  Set speed (120.0 mm/s)
  MoveL 7621 to (504.18, 492.37, 15.4) mm, rotated rx 0 ry 90 rz 0 deg; joints [-11.231, -27.866, 111.232, -15.254, -82.736, 50.97]
  Set speed (1000.0 mm/s)
  MoveL 7622 to (504.11, 492.3, 15.4) mm, rotated rx 0 ry 90 rz 0 deg; joints [-11.226, -27.867, 111.243, -15.248, -82.744, 50.967]
  Set speed (15.0 mm/s)
  Call Extruder(0.010)
  MoveL 7623 to (504.11, 491.95, 15.4) mm, rotated rx 0 ry 90 rz 0 deg; joints [-11.194, -27.869, 111.251, -15.216, -82.75, 50.961]
  Call Extruder(0.035)
  MoveL 7624 to (504.11, 490.75, 15.4) mm, rotated rx 0 ry 90 rz 0 deg; joints [-11.084, -27.873, 111.279, -15.104, -82.77, 50.943]
  Call Extruder(0.010)
  MoveL 7625 to (504.11, 490.4, 15.4) mm, rotated rx 0 ry 90 rz 0 deg; joints [-11.052, -27.874, 111.288, -15.072, -82.776, 50.937]
  Call Extruder(0.007)
  MoveL 7626 to (504.46, 490.4, 15.4) mm, rotated rx 0 ry 90 rz 0 deg; joints [-11.046, -27.868, 111.246, -15.067, -82.741, 50.946]
  Call Extruder(0.149)
  MoveL 7627 to (509.6, 490.4, 15.4) mm, rotated rx 0 ry 90 rz 0 deg; joints [-10.955, -27.767, 110.627, -14.993, -82.238, 51.071]
  Call Extruder(0.125)
  MoveL 7628 to (509.6, 494.7, 15.4) mm, rotated rx 0 ry 90 rz 0 deg; joints [-11.345, -27.75, 110.525, -15.389, -82.169, 51.141]
  Call Extruder(0.046)
  MoveL 7629 to (508.02, 494.7, 15.4) mm, rotated rx 0 ry 90 rz 0 deg; joints [-11.374, -27.781, 110.715, -15.413, -82.323, 51.102]
  Call Extruder(0.010)
  MoveL 7630 to (507.67, 494.7, 15.4) mm, rotated rx 0 ry 90 rz 0 deg; joints [-11.38, -27.788, 110.757, -15.418, -82.357, 51.093]
  Call Extruder(0.007)
  MoveL 7631 to (507.67, 495.05, 15.4) mm, rotated rx 0 ry 90 rz 0 deg; joints [-11.412, -27.787, 110.748, -15.45, -82.351, 51.099]
  Call Extruder(0.064)
  MoveL 7632 to (507.68, 497.23, 15.4) mm, rotated rx 0 ry 90 rz 0 deg; joints [-11.61, -27.778, 110.694, -15.651, -82.314, 51.135]
  Call Extruder(0.056)
  MoveL 7633 to (509.6, 497.23, 15.4) mm, rotated rx 0 ry 90 rz 0 deg; joints [-11.574, -27.739, 110.463, -15.622, -82.127, 51.183]
  Call Extruder(0.123)
  MoveL 7634 to (509.6, 501.46, 15.4) mm, rotated rx 0 ry 90 rz 0 deg; joints [-11.956, -27.722, 110.357, -16.01, -82.055, 51.254]
  Call Extruder(0.010)
  MoveL 7635 to (509.6, 501.81, 15.4) mm, rotated rx 0 ry 90 rz 0 deg; joints [-11.987, -27.72, 110.348, -16.043, -82.049, 51.26]
  Call Extruder(0.007)
  MoveL 7636 to (509.25, 501.81, 15.4) mm, rotated rx 0 ry 90 rz 0 deg; joints [-11.994, -27.727, 110.39, -16.048, -82.083, 51.251]
  Call Extruder(0.036)
  MoveL 7637 to (508.02, 501.8, 15.4) mm, rotated rx 0 ry 90 rz 0 deg; joints [-12.017, -27.752, 110.538, -16.067, -82.202, 51.22]
  Call Extruder(0.010)
  MoveL 7638 to (507.67, 501.8, 15.4) mm, rotated rx 0 ry 90 rz 0 deg; joints [-12.024, -27.759, 110.58, -16.072, -82.236, 51.211]
  Call Extruder(0.007)
  MoveL 7639 to (507.67, 502.15, 15.4) mm, rotated rx 0 ry 90 rz 0 deg; joints [-12.056, -27.758, 110.571, -16.105, -82.23, 51.217]
  Call Extruder(0.063)
  MoveL 7640 to (507.67, 504.32, 15.4) mm, rotated rx 0 ry 90 rz 0 deg; joints [-12.251, -27.748, 110.515, -16.304, -82.192, 51.254]
  Call Extruder(0.056)
  MoveL 7641 to (509.6, 504.32, 15.4) mm, rotated rx 0 ry 90 rz 0 deg; joints [-12.214, -27.709, 110.283, -16.273, -82.005, 51.304]
  Call Extruder(0.154)
  MoveL 7642 to (509.6, 509.6, 15.4) mm, rotated rx 0 ry 90 rz 0 deg; joints [-12.688, -27.685, 110.142, -16.757, -81.911, 51.397]
  Call Extruder(0.559)
  MoveL 7643 to (490.4, 509.6, 15.4) mm, rotated rx 0 ry 90 rz 0 deg; joints [-13.088, -28.05, 112.431, -17.089, -83.766, 50.877]
  MoveL 7644 to (490.4, 490.4, 15.4) mm, rotated rx 0 ry 90 rz 0 deg; joints [-11.303, -28.121, 112.922, -15.283, -84.122, 50.597]
  Call Extruder(0.130)
  MoveL 7645 to (494.86, 490.4, 15.4) mm, rotated rx 0 ry 90 rz 0 deg; joints [-11.22, -28.044, 112.392, -15.212, -83.683, 50.709]
  Call Extruder(0.010)
  MoveL 7646 to (495.21, 490.4, 15.4) mm, rotated rx 0 ry 90 rz 0 deg; joints [-11.214, -28.038, 112.351, -15.207, -83.649, 50.718]
  Call Extruder(0.007)
  MoveL 7647 to (495.21, 490.75, 15.4) mm, rotated rx 0 ry 90 rz 0 deg; joints [-11.246, -28.037, 112.342, -15.239, -83.643, 50.723]
  Call Extruder(0.035)
  MoveL 7648 to (495.21, 491.95, 15.4) mm, rotated rx 0 ry 90 rz 0 deg; joints [-11.358, -28.032, 112.314, -15.352, -83.622, 50.74]
  Call Extruder(0.010)
  MoveL 7649 to (495.21, 492.3, 15.4) mm, rotated rx 0 ry 90 rz 0 deg; joints [-11.39, -28.031, 112.306, -15.385, -83.616, 50.745]
  Call Extruder(0.007)
  MoveL 7650 to (495.56, 492.3, 15.4) mm, rotated rx 0 ry 90 rz 0 deg; joints [-11.384, -28.025, 112.264, -15.38, -83.582, 50.754]
  Call Extruder(0.061)
  MoveL 7651 to (497.67, 492.3, 15.4) mm, rotated rx 0 ry 90 rz 0 deg; joints [-11.345, -27.987, 112.014, -15.347, -83.376, 50.807]
  Call Extruder(0.055)
  MoveL 7652 to (497.67, 490.4, 15.4) mm, rotated rx 0 ry 90 rz 0 deg; joints [-11.169, -27.994, 112.059, -15.169, -83.408, 50.779]
  Call Extruder(0.116)
  MoveL 7653 to (501.67, 490.4, 15.4) mm, rotated rx 0 ry 90 rz 0 deg; joints [-11.096, -27.921, 111.581, -15.108, -83.015, 50.878]
  Call Extruder(0.036)
  MoveL 7654 to (501.67, 491.64, 15.4) mm, rotated rx 0 ry 90 rz 0 deg; joints [-11.21, -27.916, 111.551, -15.224, -82.994, 50.896]
  Call Extruder(0.019)
  MoveL 7655 to (501.67, 492.3, 15.4) mm, rotated rx 0 ry 90 rz 0 deg; joints [-11.271, -27.913, 111.535, -15.285, -82.983, 50.906]
  Call Extruder(0.061)
  MoveL 7656 to (503.76, 492.3, 15.4) mm, rotated rx 0 ry 90 rz 0 deg; joints [-11.233, -27.874, 111.285, -15.254, -82.778, 50.958]
  Call Extruder(0.007)
  MoveL 7657 to (504.11, 492.3, 15.4) mm, rotated rx 0 ry 90 rz 0 deg; joints [-11.226, -27.867, 111.243, -15.248, -82.744, 50.967]
  Set speed (120.0 mm/s)
  MoveL 7658 to (504.11, 491.95, 15.4) mm, rotated rx 0 ry 90 rz 0 deg; joints [-11.194, -27.869, 111.251, -15.216, -82.75, 50.961]
  Set speed (1000.0 mm/s)
  MoveL 7659 to (504.11, 491.9, 15.4) mm, rotated rx 0 ry 90 rz 0 deg; joints [-11.19, -27.869, 111.252, -15.211, -82.751, 50.961]
  Set speed (1000.0 mm/s)
  MoveL 7660 to (504.81, 491.9, 15.4) mm, rotated rx 0 ry 90 rz 0 deg; joints [-11.177, -27.855, 111.168, -15.201, -82.682, 50.978]
  Set speed (1000.0 mm/s)
  MoveL 7661 to (495.18, 492.33, 15.4) mm, rotated rx 0 ry 90 rz 0 deg; joints [-11.393, -28.032, 112.309, -15.388, -83.619, 50.744]
  Set speed (1000.0 mm/s)
  MoveL 7662 to (490.68, 490.68, 15.4) mm, rotated rx 0 ry 90 rz 0 deg; joints [-11.324, -28.115, 112.882, -15.304, -84.09, 50.608]
  Set speed (1000.0 mm/s)
  MoveL 7663 to (490.68, 490.68, 15.5) mm, rotated rx 0 ry 90 rz 0 deg; joints [-11.324, -28.126, 112.887, -15.305, -84.084, 50.609]
  Set speed (30.0 mm/s)
  Call Extruder(0.767)
  MoveL 7664 to (509.32, 509.32, 15.5) mm, rotated rx 0 ry 90 rz 0 deg; joints [-12.669, -27.703, 110.189, -16.736, -81.938, 51.386]
  MoveL 7665 to (509.44, 509.44, 15.5) mm, rotated rx 0 ry 90 rz 0 deg; joints [-12.677, -27.7, 110.17, -16.745, -81.924, 51.392]
  Set speed (120.0 mm/s)
  MoveL 7666 to (507.64, 504.4, 15.5) mm, rotated rx 0 ry 90 rz 0 deg; joints [-12.259, -27.759, 110.521, -16.312, -82.188, 51.256]
  Set speed (1000.0 mm/s)
  MoveL 7667 to (507.39, 502.51, 15.5) mm, rotated rx 0 ry 90 rz 0 deg; joints [-12.093, -27.772, 110.601, -16.142, -82.246, 51.217]
  Set speed (30.0 mm/s)
  Call Extruder(0.280)
  MoveL 7668 to (500.58, 509.32, 15.5) mm, rotated rx 0 ry 90 rz 0 deg; joints [-12.847, -27.876, 111.237, -16.882, -82.782, 51.152]
  Set speed (120.0 mm/s)
  MoveL 7669 to (499.42, 509.32, 15.5) mm, rotated rx 0 ry 90 rz 0 deg; joints [-12.872, -27.898, 111.375, -16.902, -82.894, 51.121]
  Set speed (30.0 mm/s)
  Call Extruder(0.360)
  MoveL 7670 to (490.68, 500.58, 15.5) mm, rotated rx 0 ry 90 rz 0 deg; joints [-12.247, -28.091, 112.643, -16.238, -83.906, 50.749]
  Set speed (120.0 mm/s)
  MoveL 7671 to (490.68, 499.42, 15.5) mm, rotated rx 0 ry 90 rz 0 deg; joints [-12.139, -28.095, 112.673, -16.129, -83.928, 50.732]
  Set speed (30.0 mm/s)
  Call Extruder(0.281)
  MoveL 7672 to (497.52, 492.58, 15.5) mm, rotated rx 0 ry 90 rz 0 deg; joints [-11.373, -28, 112.03, -15.375, -83.38, 50.808]
  Set speed (120.0 mm/s)
  MoveL 7673 to (497.89, 492.21, 15.5) mm, rotated rx 0 ry 90 rz 0 deg; joints [-11.332, -27.994, 111.995, -15.335, -83.35, 50.812]
  Set speed (30.0 mm/s)
  Call Extruder(0.063)
  MoveL 7674 to (499.42, 490.68, 15.5) mm, rotated rx 0 ry 90 rz 0 deg; joints [-11.163, -27.972, 111.848, -15.168, -83.226, 50.828]
  Set speed (120.0 mm/s)
  MoveL 7675 to (500.58, 490.68, 15.5) mm, rotated rx 0 ry 90 rz 0 deg; joints [-11.141, -27.95, 111.71, -15.151, -83.112, 50.856]
  Set speed (30.0 mm/s)
  Call Extruder(0.036)
  MoveL 7676 to (501.45, 491.55, 15.5) mm, rotated rx 0 ry 90 rz 0 deg; joints [-11.206, -27.931, 111.585, -15.219, -83.012, 50.891]
  Set speed (120.0 mm/s)
  MoveL 7677 to (502.48, 492.58, 15.5) mm, rotated rx 0 ry 90 rz 0 deg; joints [-11.282, -27.908, 111.437, -15.299, -82.894, 50.932]
  Set speed (30.0 mm/s)
  Call Extruder(0.281)
  MoveL 7678 to (509.32, 499.42, 15.5) mm, rotated rx 0 ry 90 rz 0 deg; joints [-11.777, -27.746, 110.447, -15.828, -82.112, 51.214]
  Set speed (120.0 mm/s)
  MoveL 7679 to (509.32, 500.58, 15.5) mm, rotated rx 0 ry 90 rz 0 deg; joints [-11.882, -27.741, 110.418, -15.935, -82.092, 51.234]
  Set speed (30.0 mm/s)
  Call Extruder(0.041)
  MoveL 7680 to (508.32, 501.58, 15.5) mm, rotated rx 0 ry 90 rz 0 deg; joints [-11.991, -27.757, 110.513, -16.042, -82.172, 51.225]
  MoveL 7681 to (508.2, 501.7, 15.5) mm, rotated rx 0 ry 90 rz 0 deg; joints [-12.005, -27.759, 110.525, -16.055, -82.182, 51.224]
  Set speed (120.0 mm/s)
  MoveL 7682 to (507.65, 497.2, 15.5) mm, rotated rx 0 ry 90 rz 0 deg; joints [-11.608, -27.789, 110.704, -15.649, -82.312, 51.135]
  Set speed (1000.0 mm/s)
  MoveL 7683 to (507.65, 494.61, 15.5) mm, rotated rx 0 ry 90 rz 0 deg; joints [-11.373, -27.8, 110.767, -15.41, -82.356, 51.093]
  Set speed (1000.0 mm/s)
  MoveL 7684 to (509.32, 490.68, 15.5) mm, rotated rx 0 ry 90 rz 0 deg; joints [-10.985, -27.782, 110.659, -15.023, -82.256, 51.07]
  Set speed (30.0 mm/s)
  Call Extruder(0.767)
  MoveL 7685 to (490.68, 509.32, 15.5) mm, rotated rx 0 ry 90 rz 0 deg; joints [-13.056, -28.057, 112.411, -17.058, -83.739, 50.882]
  MoveL 7686 to (490.56, 509.44, 15.5) mm, rotated rx 0 ry 90 rz 0 deg; joints [-13.07, -28.058, 112.422, -17.072, -83.749, 50.88]
  Set speed (120.0 mm/s)
  MoveL 7687 to (504.25, 492.37, 15.5) mm, rotated rx 0 ry 90 rz 0 deg; joints [-11.23, -27.875, 111.23, -15.253, -82.725, 50.973]
  Set speed (1000.0 mm/s)
  MoveL 7688 to (504.18, 492.3, 15.5) mm, rotated rx 0 ry 90 rz 0 deg; joints [-11.225, -27.876, 111.24, -15.248, -82.733, 50.97]
  Set speed (15.0 mm/s)
  Call Extruder(0.010)
  MoveL 7689 to (504.18, 491.95, 15.5) mm, rotated rx 0 ry 90 rz 0 deg; joints [-11.193, -27.878, 111.248, -15.215, -82.739, 50.964]
  Call Extruder(0.035)
  MoveL 7690 to (504.18, 490.75, 15.5) mm, rotated rx 0 ry 90 rz 0 deg; joints [-11.083, -27.882, 111.277, -15.104, -82.758, 50.946]
  Call Extruder(0.010)
  MoveL 7691 to (504.18, 490.4, 15.5) mm, rotated rx 0 ry 90 rz 0 deg; joints [-11.051, -27.884, 111.285, -15.071, -82.764, 50.94]
  Call Extruder(0.007)
  MoveL 7692 to (504.53, 490.4, 15.5) mm, rotated rx 0 ry 90 rz 0 deg; joints [-11.045, -27.877, 111.243, -15.066, -82.73, 50.949]
  Call Extruder(0.148)
  MoveL 7693 to (509.6, 490.4, 15.5) mm, rotated rx 0 ry 90 rz 0 deg; joints [-10.955, -27.777, 110.632, -14.993, -82.233, 51.072]
  Call Extruder(0.123)
  MoveL 7694 to (509.6, 494.64, 15.5) mm, rotated rx 0 ry 90 rz 0 deg; joints [-11.339, -27.76, 110.531, -15.384, -82.165, 51.141]
  Call Extruder(0.046)
  MoveL 7695 to (508.02, 494.64, 15.5) mm, rotated rx 0 ry 90 rz 0 deg; joints [-11.368, -27.792, 110.721, -15.407, -82.318, 51.102]
  Call Extruder(0.010)
  MoveL 7696 to (507.67, 494.64, 15.5) mm, rotated rx 0 ry 90 rz 0 deg; joints [-11.375, -27.799, 110.763, -15.412, -82.352, 51.094]
  Call Extruder(0.007)
  MoveL 7697 to (507.67, 494.99, 15.5) mm, rotated rx 0 ry 90 rz 0 deg; joints [-11.407, -27.798, 110.755, -15.445, -82.347, 51.099]
  Call Extruder(0.064)
  MoveL 7698 to (507.68, 497.18, 15.5) mm, rotated rx 0 ry 90 rz 0 deg; joints [-11.605, -27.789, 110.701, -15.646, -82.31, 51.135]
  Call Extruder(0.056)
  MoveL 7699 to (509.6, 497.18, 15.5) mm, rotated rx 0 ry 90 rz 0 deg; joints [-11.569, -27.75, 110.469, -15.617, -82.123, 51.183]
  Call Extruder(0.126)
  MoveL 7700 to (509.6, 501.51, 15.5) mm, rotated rx 0 ry 90 rz 0 deg; joints [-11.961, -27.732, 110.36, -16.016, -82.049, 51.257]
  Call Extruder(0.010)
  MoveL 7701 to (509.6, 501.86, 15.5) mm, rotated rx 0 ry 90 rz 0 deg; joints [-11.992, -27.73, 110.351, -16.048, -82.043, 51.263]
  Call Extruder(0.007)
  MoveL 7702 to (509.25, 501.86, 15.5) mm, rotated rx 0 ry 90 rz 0 deg; joints [-11.999, -27.737, 110.393, -16.053, -82.077, 51.254]
  Call Extruder(0.036)
  MoveL 7703 to (508.02, 501.86, 15.5) mm, rotated rx 0 ry 90 rz 0 deg; joints [-12.022, -27.762, 110.542, -16.072, -82.196, 51.222]
  Call Extruder(0.010)
  MoveL 7704 to (507.67, 501.86, 15.5) mm, rotated rx 0 ry 90 rz 0 deg; joints [-12.029, -27.769, 110.584, -16.078, -82.23, 51.213]
  Call Extruder(0.007)
  MoveL 7705 to (507.67, 502.21, 15.5) mm, rotated rx 0 ry 90 rz 0 deg; joints [-12.061, -27.768, 110.575, -16.11, -82.224, 51.219]
  Call Extruder(0.063)
  MoveL 7706 to (507.67, 504.37, 15.5) mm, rotated rx 0 ry 90 rz 0 deg; joints [-12.256, -27.758, 110.519, -16.309, -82.186, 51.256]
  Call Extruder(0.056)
  MoveL 7707 to (509.6, 504.38, 15.5) mm, rotated rx 0 ry 90 rz 0 deg; joints [-12.219, -27.719, 110.286, -16.279, -81.999, 51.306]
  Call Extruder(0.152)
  MoveL 7708 to (509.6, 509.6, 15.5) mm, rotated rx 0 ry 90 rz 0 deg; joints [-12.688, -27.696, 110.147, -16.757, -81.906, 51.399]
  Call Extruder(0.559)
  MoveL 7709 to (490.4, 509.6, 15.5) mm, rotated rx 0 ry 90 rz 0 deg; joints [-13.088, -28.06, 112.437, -17.089, -83.761, 50.878]
  MoveL 7710 to (490.4, 490.4, 15.5) mm, rotated rx 0 ry 90 rz 0 deg; joints [-11.303, -28.131, 112.927, -15.283, -84.117, 50.598]
  Call Extruder(0.128)
  MoveL 7711 to (494.81, 490.4, 15.5) mm, rotated rx 0 ry 90 rz 0 deg; joints [-11.221, -28.056, 112.404, -15.213, -83.683, 50.709]
  Call Extruder(0.010)
  MoveL 7712 to (495.16, 490.4, 15.5) mm, rotated rx 0 ry 90 rz 0 deg; joints [-11.215, -28.049, 112.363, -15.208, -83.649, 50.718]
  Call Extruder(0.007)
  MoveL 7713 to (495.16, 490.75, 15.5) mm, rotated rx 0 ry 90 rz 0 deg; joints [-11.247, -28.048, 112.354, -15.24, -83.643, 50.723]
  Call Extruder(0.035)
  MoveL 7714 to (495.15, 491.95, 15.5) mm, rotated rx 0 ry 90 rz 0 deg; joints [-11.359, -28.044, 112.326, -15.353, -83.623, 50.74]
  Call Extruder(0.010)
  MoveL 7715 to (495.16, 492.3, 15.5) mm, rotated rx 0 ry 90 rz 0 deg; joints [-11.391, -28.043, 112.318, -15.386, -83.617, 50.745]
  Call Extruder(0.007)
  MoveL 7716 to (495.5, 492.3, 15.5) mm, rotated rx 0 ry 90 rz 0 deg; joints [-11.385, -28.037, 112.276, -15.381, -83.582, 50.754]
  Call Extruder(0.061)
  MoveL 7717 to (497.61, 492.3, 15.5) mm, rotated rx 0 ry 90 rz 0 deg; joints [-11.346, -27.999, 112.026, -15.348, -83.376, 50.807]
  Call Extruder(0.055)
  MoveL 7718 to (497.61, 490.4, 15.5) mm, rotated rx 0 ry 90 rz 0 deg; joints [-11.17, -28.006, 112.071, -15.17, -83.408, 50.779]
  Call Extruder(0.120)
  MoveL 7719 to (501.73, 490.4, 15.5) mm, rotated rx 0 ry 90 rz 0 deg; joints [-11.095, -27.93, 111.578, -15.107, -83.004, 50.88]
  Call Extruder(0.037)
  MoveL 7720 to (501.73, 491.68, 15.5) mm, rotated rx 0 ry 90 rz 0 deg; joints [-11.213, -27.925, 111.548, -15.227, -82.982, 50.9]
  Call Extruder(0.018)
  MoveL 7721 to (501.74, 492.3, 15.5) mm, rotated rx 0 ry 90 rz 0 deg; joints [-11.27, -27.923, 111.533, -15.285, -82.972, 50.909]
  Call Extruder(0.061)
  MoveL 7722 to (503.83, 492.3, 15.5) mm, rotated rx 0 ry 90 rz 0 deg; joints [-11.232, -27.883, 111.282, -15.253, -82.767, 50.961]
  Call Extruder(0.007)
  MoveL 7723 to (504.18, 492.3, 15.5) mm, rotated rx 0 ry 90 rz 0 deg; joints [-11.225, -27.876, 111.24, -15.248, -82.733, 50.97]
  Set speed (120.0 mm/s)
  MoveL 7724 to (504.18, 491.95, 15.5) mm, rotated rx 0 ry 90 rz 0 deg; joints [-11.193, -27.878, 111.248, -15.215, -82.739, 50.964]
  Set speed (1000.0 mm/s)
  MoveL 7725 to (504.18, 491.9, 15.5) mm, rotated rx 0 ry 90 rz 0 deg; joints [-11.189, -27.878, 111.249, -15.211, -82.739, 50.964]
  Set speed (1000.0 mm/s)
  MoveL 7726 to (504.88, 491.9, 15.5) mm, rotated rx 0 ry 90 rz 0 deg; joints [-11.176, -27.865, 111.165, -15.2, -82.671, 50.981]
  Set speed (1000.0 mm/s)
  MoveL 7727 to (495.13, 492.33, 15.5) mm, rotated rx 0 ry 90 rz 0 deg; joints [-11.394, -28.043, 112.32, -15.389, -83.619, 50.745]
  Set speed (1000.0 mm/s)
  MoveL 7728 to (490.68, 490.68, 15.5) mm, rotated rx 0 ry 90 rz 0 deg; joints [-11.324, -28.126, 112.887, -15.305, -84.084, 50.609]
  Set speed (1000.0 mm/s)
  MoveL 7729 to (490.68, 490.68, 15.6) mm, rotated rx 0 ry 90 rz 0 deg; joints [-11.324, -28.136, 112.893, -15.305, -84.079, 50.61]
  Set speed (30.0 mm/s)
  Call Extruder(0.767)
  MoveL 7730 to (509.32, 509.32, 15.6) mm, rotated rx 0 ry 90 rz 0 deg; joints [-12.669, -27.713, 110.194, -16.736, -81.933, 51.388]
  MoveL 7731 to (509.44, 509.44, 15.6) mm, rotated rx 0 ry 90 rz 0 deg; joints [-12.677, -27.71, 110.176, -16.745, -81.919, 51.393]
  Set speed (120.0 mm/s)
  MoveL 7732 to (507.64, 504.46, 15.6) mm, rotated rx 0 ry 90 rz 0 deg; joints [-12.264, -27.769, 110.525, -16.317, -82.182, 51.258]
  Set speed (1000.0 mm/s)
  MoveL 7733 to (507.39, 502.51, 15.6) mm, rotated rx 0 ry 90 rz 0 deg; joints [-12.093, -27.783, 110.606, -16.142, -82.241, 51.219]
  Set speed (30.0 mm/s)
  Call Extruder(0.280)
  MoveL 7734 to (500.58, 509.32, 15.6) mm, rotated rx 0 ry 90 rz 0 deg; joints [-12.847, -27.886, 111.242, -16.882, -82.777, 51.154]
  Set speed (120.0 mm/s)
  MoveL 7735 to (499.42, 509.32, 15.6) mm, rotated rx 0 ry 90 rz 0 deg; joints [-12.872, -27.909, 111.38, -16.902, -82.889, 51.123]
  Set speed (30.0 mm/s)
  Call Extruder(0.360)
  MoveL 7736 to (490.68, 500.58, 15.6) mm, rotated rx 0 ry 90 rz 0 deg; joints [-12.247, -28.101, 112.648, -16.238, -83.901, 50.751]
  Set speed (120.0 mm/s)
  MoveL 7737 to (490.68, 499.42, 15.6) mm, rotated rx 0 ry 90 rz 0 deg; joints [-12.139, -28.105, 112.678, -16.129, -83.923, 50.734]
  Set speed (30.0 mm/s)
  Call Extruder(0.281)
  MoveL 7738 to (497.52, 492.58, 15.6) mm, rotated rx 0 ry 90 rz 0 deg; joints [-11.373, -28.01, 112.035, -15.376, -83.375, 50.81]
  Set speed (120.0 mm/s)
  MoveL 7739 to (497.83, 492.27, 15.6) mm, rotated rx 0 ry 90 rz 0 deg; joints [-11.338, -28.006, 112.005, -15.341, -83.349, 50.813]
  Set speed (30.0 mm/s)
  Call Extruder(0.065)
  MoveL 7740 to (499.42, 490.68, 15.6) mm, rotated rx 0 ry 90 rz 0 deg; joints [-11.163, -27.982, 111.853, -15.168, -83.221, 50.829]
  Set speed (120.0 mm/s)
  MoveL 7741 to (500.58, 490.68, 15.6) mm, rotated rx 0 ry 90 rz 0 deg; joints [-11.141, -27.961, 111.715, -15.151, -83.107, 50.858]
  Set speed (30.0 mm/s)
  Call Extruder(0.039)
  MoveL 7742 to (501.51, 491.62, 15.6) mm, rotated rx 0 ry 90 rz 0 deg; joints [-11.211, -27.94, 111.581, -15.224, -83, 50.895]
  Set speed (120.0 mm/s)
  MoveL 7743 to (502.48, 492.58, 15.6) mm, rotated rx 0 ry 90 rz 0 deg; joints [-11.282, -27.918, 111.442, -15.299, -82.889, 50.934]
  Set speed (30.0 mm/s)
  Call Extruder(0.281)
  MoveL 7744 to (509.32, 499.42, 15.6) mm, rotated rx 0 ry 90 rz 0 deg; joints [-11.777, -27.757, 110.452, -15.828, -82.107, 51.216]
  Set speed (120.0 mm/s)
  MoveL 7745 to (509.32, 500.58, 15.6) mm, rotated rx 0 ry 90 rz 0 deg; joints [-11.882, -27.752, 110.423, -15.935, -82.087, 51.235]
  Set speed (30.0 mm/s)
  Call Extruder(0.043)
  MoveL 7746 to (508.26, 501.63, 15.6) mm, rotated rx 0 ry 90 rz 0 deg; joints [-11.997, -27.769, 110.523, -16.048, -82.171, 51.226]
  MoveL 7747 to (508.14, 501.76, 15.6) mm, rotated rx 0 ry 90 rz 0 deg; joints [-12.011, -27.771, 110.535, -16.061, -82.181, 51.225]
  Set speed (120.0 mm/s)
  MoveL 7748 to (507.65, 497.14, 15.6) mm, rotated rx 0 ry 90 rz 0 deg; joints [-11.602, -27.8, 110.71, -15.644, -82.308, 51.136]
  Set speed (1000.0 mm/s)
  MoveL 7749 to (507.65, 494.55, 15.6) mm, rotated rx 0 ry 90 rz 0 deg; joints [-11.367, -27.81, 110.774, -15.405, -82.351, 51.093]
  Set speed (1000.0 mm/s)
  MoveL 7750 to (509.32, 490.68, 15.6) mm, rotated rx 0 ry 90 rz 0 deg; joints [-10.985, -27.792, 110.665, -15.023, -82.251, 51.071]
  Set speed (30.0 mm/s)
  Call Extruder(0.767)
  MoveL 7751 to (490.68, 509.32, 15.6) mm, rotated rx 0 ry 90 rz 0 deg; joints [-13.056, -28.067, 112.416, -17.058, -83.734, 50.883]
  MoveL 7752 to (490.56, 509.44, 15.6) mm, rotated rx 0 ry 90 rz 0 deg; joints [-13.07, -28.069, 112.428, -17.072, -83.743, 50.882]
  Set speed (120.0 mm/s)
  MoveL 7753 to (504.31, 492.37, 15.6) mm, rotated rx 0 ry 90 rz 0 deg; joints [-11.229, -27.884, 111.227, -15.252, -82.713, 50.976]
  Set speed (1000.0 mm/s)
  MoveL 7754 to (504.24, 492.3, 15.6) mm, rotated rx 0 ry 90 rz 0 deg; joints [-11.224, -27.886, 111.237, -15.247, -82.721, 50.973]
  Set speed (15.0 mm/s)
  Call Extruder(0.010)
  MoveL 7755 to (504.24, 491.95, 15.6) mm, rotated rx 0 ry 90 rz 0 deg; joints [-11.192, -27.887, 111.246, -15.215, -82.727, 50.968]
  Call Extruder(0.035)
  MoveL 7756 to (504.24, 490.75, 15.6) mm, rotated rx 0 ry 90 rz 0 deg; joints [-11.082, -27.892, 111.274, -15.103, -82.747, 50.949]
  Call Extruder(0.010)
  MoveL 7757 to (504.24, 490.4, 15.6) mm, rotated rx 0 ry 90 rz 0 deg; joints [-11.05, -27.893, 111.282, -15.07, -82.753, 50.943]
  Call Extruder(0.007)
  MoveL 7758 to (504.59, 490.4, 15.6) mm, rotated rx 0 ry 90 rz 0 deg; joints [-11.044, -27.886, 111.24, -15.065, -82.718, 50.952]
  Call Extruder(0.146)
  MoveL 7759 to (509.6, 490.4, 15.6) mm, rotated rx 0 ry 90 rz 0 deg; joints [-10.955, -27.788, 110.637, -14.993, -82.228, 51.074]
  Call Extruder(0.122)
  MoveL 7760 to (509.6, 494.58, 15.6) mm, rotated rx 0 ry 90 rz 0 deg; joints [-11.334, -27.771, 110.538, -15.378, -82.16, 51.142]
  Call Extruder(0.056)
  MoveL 7761 to (507.67, 494.58, 15.6) mm, rotated rx 0 ry 90 rz 0 deg; joints [-11.369, -27.81, 110.77, -15.407, -82.348, 51.094]
  Call Extruder(0.056)
  MoveL 7762 to (507.67, 496.51, 15.6) mm, rotated rx 0 ry 90 rz 0 deg; joints [-11.545, -27.802, 110.723, -15.585, -82.316, 51.126]
  Call Extruder(0.003)
  MoveL 7763 to (507.67, 496.61, 15.6) mm, rotated rx 0 ry 90 rz 0 deg; joints [-11.554, -27.802, 110.72, -15.595, -82.315, 51.127]
  Call Extruder(0.015)
  MoveL 7764 to (507.68, 497.12, 15.6) mm, rotated rx 0 ry 90 rz 0 deg; joints [-11.599, -27.799, 110.707, -15.641, -82.306, 51.136]
  Call Extruder(0.003)
  MoveL 7765 to (507.78, 497.12, 15.6) mm, rotated rx 0 ry 90 rz 0 deg; joints [-11.598, -27.798, 110.696, -15.639, -82.296, 51.138]
  Call Extruder(0.053)
  MoveL 7766 to (509.6, 497.12, 15.6) mm, rotated rx 0 ry 90 rz 0 deg; joints [-11.564, -27.761, 110.476, -15.612, -82.118, 51.184]
  Call Extruder(0.130)
  MoveL 7767 to (509.6, 501.57, 15.6) mm, rotated rx 0 ry 90 rz 0 deg; joints [-11.966, -27.742, 110.364, -16.021, -82.043, 51.259]
  Call Extruder(0.010)
  MoveL 7768 to (509.6, 501.92, 15.6) mm, rotated rx 0 ry 90 rz 0 deg; joints [-11.997, -27.74, 110.355, -16.053, -82.037, 51.265]
  Call Extruder(0.007)
  MoveL 7769 to (509.25, 501.92, 15.6) mm, rotated rx 0 ry 90 rz 0 deg; joints [-12.004, -27.748, 110.397, -16.059, -82.071, 51.256]
  Call Extruder(0.036)
  MoveL 7770 to (508.02, 501.91, 15.6) mm, rotated rx 0 ry 90 rz 0 deg; joints [-12.027, -27.772, 110.545, -16.077, -82.19, 51.225]
  Call Extruder(0.010)
  MoveL 7771 to (507.67, 501.91, 15.6) mm, rotated rx 0 ry 90 rz 0 deg; joints [-12.034, -27.78, 110.587, -16.083, -82.224, 51.216]
  Call Extruder(0.007)
  MoveL 7772 to (507.67, 502.26, 15.6) mm, rotated rx 0 ry 90 rz 0 deg; joints [-12.066, -27.778, 110.578, -16.115, -82.218, 51.222]
  Call Extruder(0.063)
  MoveL 7773 to (507.67, 504.43, 15.6) mm, rotated rx 0 ry 90 rz 0 deg; joints [-12.261, -27.769, 110.522, -16.314, -82.18, 51.259]
  Call Extruder(0.056)
  MoveL 7774 to (509.6, 504.43, 15.6) mm, rotated rx 0 ry 90 rz 0 deg; joints [-12.224, -27.729, 110.29, -16.284, -81.993, 51.309]
  Call Extruder(0.150)
  MoveL 7775 to (509.6, 509.6, 15.6) mm, rotated rx 0 ry 90 rz 0 deg; joints [-12.688, -27.706, 110.152, -16.757, -81.901, 51.4]
  Call Extruder(0.559)
  MoveL 7776 to (490.4, 509.6, 15.6) mm, rotated rx 0 ry 90 rz 0 deg; joints [-13.088, -28.071, 112.442, -17.089, -83.755, 50.88]
  MoveL 7777 to (490.4, 490.4, 15.6) mm, rotated rx 0 ry 90 rz 0 deg; joints [-11.303, -28.142, 112.932, -15.283, -84.111, 50.6]
  Call Extruder(0.127)
  MoveL 7778 to (494.75, 490.4, 15.6) mm, rotated rx 0 ry 90 rz 0 deg; joints [-11.222, -28.067, 112.416, -15.214, -83.683, 50.709]
  Call Extruder(0.010)
  MoveL 7779 to (495.1, 490.4, 15.6) mm, rotated rx 0 ry 90 rz 0 deg; joints [-11.216, -28.061, 112.374, -15.209, -83.649, 50.718]
  Call Extruder(0.007)
  MoveL 7780 to (495.1, 490.75, 15.6) mm, rotated rx 0 ry 90 rz 0 deg; joints [-11.248, -28.06, 112.366, -15.241, -83.643, 50.723]
  Call Extruder(0.035)
  MoveL 7781 to (495.1, 491.95, 15.6) mm, rotated rx 0 ry 90 rz 0 deg; joints [-11.36, -28.056, 112.338, -15.355, -83.623, 50.74]
  Call Extruder(0.010)
  MoveL 7782 to (495.1, 492.3, 15.6) mm, rotated rx 0 ry 90 rz 0 deg; joints [-11.392, -28.054, 112.33, -15.387, -83.617, 50.745]
  Call Extruder(0.007)
  MoveL 7783 to (495.45, 492.3, 15.6) mm, rotated rx 0 ry 90 rz 0 deg; joints [-11.386, -28.048, 112.288, -15.382, -83.583, 50.754]
  Call Extruder(0.061)
  MoveL 7784 to (497.55, 492.3, 15.6) mm, rotated rx 0 ry 90 rz 0 deg; joints [-11.347, -28.011, 112.037, -15.349, -83.376, 50.807]
  Call Extruder(0.055)
  MoveL 7785 to (497.55, 490.4, 15.6) mm, rotated rx 0 ry 90 rz 0 deg; joints [-11.171, -28.017, 112.082, -15.171, -83.408, 50.779]
  Call Extruder(0.123)
  MoveL 7786 to (501.8, 490.4, 15.6) mm, rotated rx 0 ry 90 rz 0 deg; joints [-11.094, -27.939, 111.576, -15.107, -82.992, 50.883]
  Call Extruder(0.038)
  MoveL 7787 to (501.8, 491.72, 15.6) mm, rotated rx 0 ry 90 rz 0 deg; joints [-11.215, -27.934, 111.544, -15.23, -82.97, 50.904]
  Call Extruder(0.017)
  MoveL 7788 to (501.8, 492.3, 15.6) mm, rotated rx 0 ry 90 rz 0 deg; joints [-11.269, -27.932, 111.53, -15.284, -82.96, 50.912]
  Call Extruder(0.061)
  MoveL 7789 to (503.89, 492.3, 15.6) mm, rotated rx 0 ry 90 rz 0 deg; joints [-11.23, -27.893, 111.279, -15.252, -82.755, 50.964]
  Call Extruder(0.007)
  MoveL 7790 to (504.24, 492.3, 15.6) mm, rotated rx 0 ry 90 rz 0 deg; joints [-11.224, -27.886, 111.237, -15.247, -82.721, 50.973]
  Set speed (120.0 mm/s)
  MoveL 7791 to (504.24, 491.95, 15.6) mm, rotated rx 0 ry 90 rz 0 deg; joints [-11.192, -27.887, 111.246, -15.215, -82.727, 50.968]
  Set speed (1000.0 mm/s)
  MoveL 7792 to (504.24, 491.9, 15.6) mm, rotated rx 0 ry 90 rz 0 deg; joints [-11.187, -27.887, 111.247, -15.21, -82.728, 50.967]
  Set speed (1000.0 mm/s)
  MoveL 7793 to (504.94, 491.9, 15.6) mm, rotated rx 0 ry 90 rz 0 deg; joints [-11.175, -27.874, 111.163, -15.2, -82.659, 50.984]
  Set speed (1000.0 mm/s)
  MoveL 7794 to (495.07, 492.33, 15.6) mm, rotated rx 0 ry 90 rz 0 deg; joints [-11.396, -28.055, 112.332, -15.39, -83.619, 50.745]
  Set speed (1000.0 mm/s)
  MoveL 7795 to (490.68, 490.68, 15.6) mm, rotated rx 0 ry 90 rz 0 deg; joints [-11.324, -28.136, 112.893, -15.305, -84.079, 50.61]
  Set speed (1000.0 mm/s)
  MoveL 7796 to (490.68, 490.68, 15.7) mm, rotated rx 0 ry 90 rz 0 deg; joints [-11.324, -28.147, 112.898, -15.305, -84.074, 50.612]
  Set speed (30.0 mm/s)
  Call Extruder(0.767)
  MoveL 7797 to (509.32, 509.32, 15.7) mm, rotated rx 0 ry 90 rz 0 deg; joints [-12.669, -27.724, 110.199, -16.736, -81.928, 51.389]
  MoveL 7798 to (509.44, 509.44, 15.7) mm, rotated rx 0 ry 90 rz 0 deg; joints [-12.677, -27.72, 110.181, -16.746, -81.914, 51.395]
  Set speed (120.0 mm/s)
  MoveL 7799 to (507.64, 504.51, 15.7) mm, rotated rx 0 ry 90 rz 0 deg; joints [-12.27, -27.779, 110.529, -16.323, -82.176, 51.261]
  Set speed (1000.0 mm/s)
  MoveL 7800 to (507.39, 502.51, 15.7) mm, rotated rx 0 ry 90 rz 0 deg; joints [-12.093, -27.793, 110.611, -16.142, -82.236, 51.22]
  Set speed (30.0 mm/s)
  Call Extruder(0.280)
  MoveL 7801 to (500.58, 509.32, 15.7) mm, rotated rx 0 ry 90 rz 0 deg; joints [-12.847, -27.897, 111.247, -16.883, -82.771, 51.156]
  Set speed (120.0 mm/s)
  MoveL 7802 to (499.42, 509.32, 15.7) mm, rotated rx 0 ry 90 rz 0 deg; joints [-12.872, -27.919, 111.385, -16.903, -82.883, 51.124]
  Set speed (30.0 mm/s)
  Call Extruder(0.360)
  MoveL 7803 to (490.68, 500.58, 15.7) mm, rotated rx 0 ry 90 rz 0 deg; joints [-12.247, -28.112, 112.653, -16.238, -83.896, 50.752]
  Set speed (120.0 mm/s)
  MoveL 7804 to (490.68, 499.42, 15.7) mm, rotated rx 0 ry 90 rz 0 deg; joints [-12.139, -28.116, 112.683, -16.129, -83.917, 50.735]
  Set speed (30.0 mm/s)
  Call Extruder(0.281)
  MoveL 7805 to (497.52, 492.58, 15.7) mm, rotated rx 0 ry 90 rz 0 deg; joints [-11.373, -28.021, 112.04, -15.376, -83.37, 50.811]
  Set speed (120.0 mm/s)
  MoveL 7806 to (497.77, 492.32, 15.7) mm, rotated rx 0 ry 90 rz 0 deg; joints [-11.345, -28.017, 112.016, -15.348, -83.349, 50.814]
  Set speed (30.0 mm/s)
  Call Extruder(0.068)
  MoveL 7807 to (499.42, 490.68, 15.7) mm, rotated rx 0 ry 90 rz 0 deg; joints [-11.163, -27.993, 111.858, -15.169, -83.215, 50.83]
  Set speed (120.0 mm/s)
  MoveL 7808 to (500.58, 490.68, 15.7) mm, rotated rx 0 ry 90 rz 0 deg; joints [-11.142, -27.972, 111.72, -15.151, -83.102, 50.859]
  Set speed (30.0 mm/s)
  Call Extruder(0.041)
  MoveL 7809 to (501.58, 491.68, 15.7) mm, rotated rx 0 ry 90 rz 0 deg; joints [-11.215, -27.949, 111.577, -15.229, -82.987, 50.899]
  Set speed (120.0 mm/s)
  MoveL 7810 to (502.48, 492.58, 15.7) mm, rotated rx 0 ry 90 rz 0 deg; joints [-11.282, -27.929, 111.447, -15.3, -82.884, 50.935]
  Set speed (30.0 mm/s)
  Call Extruder(0.281)
  MoveL 7811 to (509.32, 499.42, 15.7) mm, rotated rx 0 ry 90 rz 0 deg; joints [-11.777, -27.767, 110.457, -15.828, -82.102, 51.217]
  Set speed (120.0 mm/s)
  MoveL 7812 to (509.32, 500.58, 15.7) mm, rotated rx 0 ry 90 rz 0 deg; joints [-11.882, -27.762, 110.428, -15.935, -82.082, 51.237]
  Set speed (30.0 mm/s)
  Call Extruder(0.046)
  MoveL 7813 to (508.21, 501.69, 15.7) mm, rotated rx 0 ry 90 rz 0 deg; joints [-12.003, -27.78, 110.534, -16.054, -82.171, 51.227]
  MoveL 7814 to (508.08, 501.81, 15.7) mm, rotated rx 0 ry 90 rz 0 deg; joints [-12.017, -27.782, 110.545, -16.067, -82.18, 51.226]
  Set speed (120.0 mm/s)
  MoveL 7815 to (507.63, 496.58, 15.7) mm, rotated rx 0 ry 90 rz 0 deg; joints [-11.551, -27.813, 110.731, -15.592, -82.314, 51.127]
  Set speed (1000.0 mm/s)
  MoveL 7816 to (507.65, 494.49, 15.7) mm, rotated rx 0 ry 90 rz 0 deg; joints [-11.362, -27.821, 110.781, -15.4, -82.347, 51.093]
  Set speed (1000.0 mm/s)
  MoveL 7817 to (509.32, 490.68, 15.7) mm, rotated rx 0 ry 90 rz 0 deg; joints [-10.985, -27.803, 110.67, -15.023, -82.246, 51.073]
  Set speed (30.0 mm/s)
  Call Extruder(0.767)
  MoveL 7818 to (490.68, 509.32, 15.7) mm, rotated rx 0 ry 90 rz 0 deg; joints [-13.056, -28.078, 112.422, -17.058, -83.729, 50.885]
  MoveL 7819 to (490.56, 509.44, 15.7) mm, rotated rx 0 ry 90 rz 0 deg; joints [-13.07, -28.08, 112.433, -17.072, -83.738, 50.883]
  Set speed (120.0 mm/s)
  MoveL 7820 to (504.38, 492.37, 15.7) mm, rotated rx 0 ry 90 rz 0 deg; joints [-11.228, -27.893, 111.225, -15.252, -82.702, 50.979]
  Set speed (1000.0 mm/s)
  MoveL 7821 to (504.31, 492.3, 15.7) mm, rotated rx 0 ry 90 rz 0 deg; joints [-11.223, -27.895, 111.235, -15.246, -82.71, 50.976]
  Set speed (15.0 mm/s)
  Call Extruder(0.010)
  MoveL 7822 to (504.31, 491.95, 15.7) mm, rotated rx 0 ry 90 rz 0 deg; joints [-11.191, -27.896, 111.243, -15.214, -82.715, 50.971]
  Call Extruder(0.035)
  MoveL 7823 to (504.3, 490.75, 15.7) mm, rotated rx 0 ry 90 rz 0 deg; joints [-11.081, -27.901, 111.272, -15.102, -82.735, 50.952]
  Call Extruder(0.010)
  MoveL 7824 to (504.31, 490.4, 15.7) mm, rotated rx 0 ry 90 rz 0 deg; joints [-11.049, -27.902, 111.28, -15.07, -82.741, 50.946]
  Call Extruder(0.007)
  MoveL 7825 to (504.66, 490.4, 15.7) mm, rotated rx 0 ry 90 rz 0 deg; joints [-11.043, -27.896, 111.238, -15.065, -82.707, 50.955]
  Call Extruder(0.144)
  MoveL 7826 to (509.6, 490.4, 15.7) mm, rotated rx 0 ry 90 rz 0 deg; joints [-10.955, -27.798, 110.642, -14.993, -82.223, 51.075]
  Call Extruder(0.120)
  MoveL 7827 to (509.6, 494.52, 15.7) mm, rotated rx 0 ry 90 rz 0 deg; joints [-11.329, -27.782, 110.544, -15.373, -82.156, 51.142]
  Call Extruder(0.056)
  MoveL 7828 to (507.67, 494.52, 15.7) mm, rotated rx 0 ry 90 rz 0 deg; joints [-11.364, -27.821, 110.776, -15.402, -82.344, 51.095]
  Call Extruder(0.057)
  MoveL 7829 to (507.67, 496.47, 15.7) mm, rotated rx 0 ry 90 rz 0 deg; joints [-11.541, -27.813, 110.729, -15.581, -82.312, 51.126]
  Call Extruder(0.003)
  MoveL 7830 to (507.67, 496.58, 15.7) mm, rotated rx 0 ry 90 rz 0 deg; joints [-11.551, -27.812, 110.726, -15.592, -82.31, 51.128]
  Call Extruder(0.014)
  MoveL 7831 to (507.68, 497.06, 15.7) mm, rotated rx 0 ry 90 rz 0 deg; joints [-11.594, -27.81, 110.714, -15.636, -82.301, 51.136]
  Call Extruder(0.003)
  MoveL 7832 to (507.79, 497.06, 15.7) mm, rotated rx 0 ry 90 rz 0 deg; joints [-11.592, -27.808, 110.701, -15.634, -82.291, 51.139]
  Call Extruder(0.053)
  MoveL 7833 to (509.6, 497.06, 15.7) mm, rotated rx 0 ry 90 rz 0 deg; joints [-11.558, -27.772, 110.482, -15.607, -82.114, 51.184]
  Call Extruder(0.133)
  MoveL 7834 to (509.6, 501.62, 15.7) mm, rotated rx 0 ry 90 rz 0 deg; joints [-11.971, -27.752, 110.368, -16.026, -82.037, 51.262]
  Call Extruder(0.010)
  MoveL 7835 to (509.6, 501.97, 15.7) mm, rotated rx 0 ry 90 rz 0 deg; joints [-12.002, -27.751, 110.359, -16.059, -82.031, 51.268]
  Call Extruder(0.007)
  MoveL 7836 to (509.25, 501.97, 15.7) mm, rotated rx 0 ry 90 rz 0 deg; joints [-12.009, -27.758, 110.401, -16.064, -82.065, 51.259]
  Call Extruder(0.036)
  MoveL 7837 to (508.02, 501.97, 15.7) mm, rotated rx 0 ry 90 rz 0 deg; joints [-12.032, -27.783, 110.549, -16.083, -82.184, 51.227]
  Call Extruder(0.010)
  MoveL 7838 to (507.67, 501.97, 15.7) mm, rotated rx 0 ry 90 rz 0 deg; joints [-12.039, -27.79, 110.591, -16.088, -82.218, 51.218]
  Call Extruder(0.007)
  MoveL 7839 to (507.67, 502.32, 15.7) mm, rotated rx 0 ry 90 rz 0 deg; joints [-12.071, -27.788, 110.582, -16.121, -82.212, 51.224]
  Call Extruder(0.063)
  MoveL 7840 to (507.67, 504.49, 15.7) mm, rotated rx 0 ry 90 rz 0 deg; joints [-12.266, -27.779, 110.526, -16.32, -82.174, 51.261]
  Call Extruder(0.056)
  MoveL 7841 to (509.6, 504.49, 15.7) mm, rotated rx 0 ry 90 rz 0 deg; joints [-12.229, -27.74, 110.293, -16.289, -81.987, 51.311]
  Call Extruder(0.149)
  MoveL 7842 to (509.6, 509.6, 15.7) mm, rotated rx 0 ry 90 rz 0 deg; joints [-12.688, -27.716, 110.157, -16.757, -81.896, 51.402]
  Call Extruder(0.559)
  MoveL 7843 to (490.4, 509.6, 15.7) mm, rotated rx 0 ry 90 rz 0 deg; joints [-13.088, -28.082, 112.447, -17.09, -83.75, 50.882]
  MoveL 7844 to (490.4, 490.4, 15.7) mm, rotated rx 0 ry 90 rz 0 deg; joints [-11.303, -28.153, 112.937, -15.283, -84.106, 50.601]
  Call Extruder(0.125)
  MoveL 7845 to (494.69, 490.4, 15.7) mm, rotated rx 0 ry 90 rz 0 deg; joints [-11.223, -28.079, 112.428, -15.215, -83.684, 50.709]
  Call Extruder(0.000)
  MoveL 7846 to (494.7, 490.4, 15.7) mm, rotated rx 0 ry 90 rz 0 deg; joints [-11.223, -28.079, 112.428, -15.215, -83.684, 50.709]
  Call Extruder(0.010)
  MoveL 7847 to (495.05, 490.4, 15.7) mm, rotated rx 0 ry 90 rz 0 deg; joints [-11.217, -28.073, 112.386, -15.21, -83.649, 50.718]
  Call Extruder(0.007)
  MoveL 7848 to (495.05, 490.75, 15.7) mm, rotated rx 0 ry 90 rz 0 deg; joints [-11.249, -28.071, 112.378, -15.243, -83.643, 50.723]
  Call Extruder(0.000)
  MoveL 7849 to (495.05, 490.75, 15.7) mm, rotated rx 0 ry 90 rz 0 deg; joints [-11.249, -28.071, 112.378, -15.243, -83.643, 50.723]
  Call Extruder(0.035)
  MoveL 7850 to (495.04, 491.95, 15.7) mm, rotated rx 0 ry 90 rz 0 deg; joints [-11.361, -28.067, 112.35, -15.356, -83.623, 50.74]
  Call Extruder(0.010)
  MoveL 7851 to (495.04, 492.3, 15.7) mm, rotated rx 0 ry 90 rz 0 deg; joints [-11.393, -28.066, 112.342, -15.388, -83.617, 50.745]
  Call Extruder(0.007)
  MoveL 7852 to (495.39, 492.3, 15.7) mm, rotated rx 0 ry 90 rz 0 deg; joints [-11.387, -28.06, 112.3, -15.383, -83.583, 50.754]
  Call Extruder(0.061)
  MoveL 7853 to (497.5, 492.3, 15.7) mm, rotated rx 0 ry 90 rz 0 deg; joints [-11.348, -28.022, 112.049, -15.35, -83.376, 50.807]
  Call Extruder(0.055)
  MoveL 7854 to (497.5, 490.4, 15.7) mm, rotated rx 0 ry 90 rz 0 deg; joints [-11.172, -28.029, 112.094, -15.172, -83.408, 50.779]
  Call Extruder(0.127)
  MoveL 7855 to (501.86, 490.4, 15.7) mm, rotated rx 0 ry 90 rz 0 deg; joints [-11.093, -27.949, 111.573, -15.106, -82.981, 50.886]
  Call Extruder(0.040)
  MoveL 7856 to (501.86, 491.76, 15.7) mm, rotated rx 0 ry 90 rz 0 deg; joints [-11.218, -27.944, 111.541, -15.233, -82.958, 50.907]
  Call Extruder(0.016)
  MoveL 7857 to (501.86, 492.3, 15.7) mm, rotated rx 0 ry 90 rz 0 deg; joints [-11.267, -27.942, 111.528, -15.283, -82.949, 50.916]
  Call Extruder(0.061)
  MoveL 7858 to (503.96, 492.3, 15.7) mm, rotated rx 0 ry 90 rz 0 deg; joints [-11.229, -27.902, 111.277, -15.251, -82.744, 50.967]
  Call Extruder(0.007)
  MoveL 7859 to (504.31, 492.3, 15.7) mm, rotated rx 0 ry 90 rz 0 deg; joints [-11.223, -27.895, 111.235, -15.246, -82.71, 50.976]
  Set speed (120.0 mm/s)
  MoveL 7860 to (504.31, 491.95, 15.7) mm, rotated rx 0 ry 90 rz 0 deg; joints [-11.191, -27.896, 111.243, -15.214, -82.715, 50.971]
  Set speed (1000.0 mm/s)
  MoveL 7861 to (504.31, 491.9, 15.7) mm, rotated rx 0 ry 90 rz 0 deg; joints [-11.186, -27.897, 111.244, -15.209, -82.716, 50.97]
  Set speed (1000.0 mm/s)
  MoveL 7862 to (505.01, 491.9, 15.7) mm, rotated rx 0 ry 90 rz 0 deg; joints [-11.174, -27.883, 111.16, -15.199, -82.648, 50.987]
  Set speed (1000.0 mm/s)
  MoveL 7863 to (495.01, 492.33, 15.7) mm, rotated rx 0 ry 90 rz 0 deg; joints [-11.397, -28.066, 112.344, -15.392, -83.619, 50.745]
  Set speed (1000.0 mm/s)
  MoveL 7864 to (490.68, 490.68, 15.7) mm, rotated rx 0 ry 90 rz 0 deg; joints [-11.324, -28.147, 112.898, -15.305, -84.074, 50.612]
  Set speed (1000.0 mm/s)
  MoveL 7865 to (490.68, 490.68, 15.8) mm, rotated rx 0 ry 90 rz 0 deg; joints [-11.324, -28.158, 112.903, -15.305, -84.068, 50.613]
  Set speed (30.0 mm/s)
  Call Extruder(0.767)
  MoveL 7866 to (509.32, 509.32, 15.8) mm, rotated rx 0 ry 90 rz 0 deg; joints [-12.669, -27.734, 110.204, -16.737, -81.923, 51.391]
  MoveL 7867 to (509.44, 509.44, 15.8) mm, rotated rx 0 ry 90 rz 0 deg; joints [-12.677, -27.731, 110.186, -16.746, -81.909, 51.396]
  Set speed (120.0 mm/s)
  MoveL 7868 to (507.64, 504.57, 15.8) mm, rotated rx 0 ry 90 rz 0 deg; joints [-12.274, -27.79, 110.532, -16.328, -82.17, 51.264]
  Set speed (1000.0 mm/s)
  MoveL 7869 to (507.39, 502.51, 15.8) mm, rotated rx 0 ry 90 rz 0 deg; joints [-12.093, -27.804, 110.616, -16.143, -82.231, 51.222]
  Set speed (30.0 mm/s)
  Call Extruder(0.280)
  MoveL 7870 to (500.58, 509.32, 15.8) mm, rotated rx 0 ry 90 rz 0 deg; joints [-12.847, -27.908, 111.252, -16.883, -82.766, 51.157]
  Set speed (120.0 mm/s)
  MoveL 7871 to (499.42, 509.32, 15.8) mm, rotated rx 0 ry 90 rz 0 deg; joints [-12.872, -27.93, 111.39, -16.903, -82.878, 51.126]
  Set speed (30.0 mm/s)
  Call Extruder(0.360)
  MoveL 7872 to (490.68, 500.58, 15.8) mm, rotated rx 0 ry 90 rz 0 deg; joints [-12.247, -28.122, 112.658, -16.239, -83.89, 50.754]
  Set speed (120.0 mm/s)
  MoveL 7873 to (490.68, 499.42, 15.8) mm, rotated rx 0 ry 90 rz 0 deg; joints [-12.139, -28.127, 112.688, -16.129, -83.912, 50.737]
  Set speed (30.0 mm/s)
  Call Extruder(0.281)
  MoveL 7874 to (497.52, 492.58, 15.8) mm, rotated rx 0 ry 90 rz 0 deg; joints [-11.373, -28.031, 112.045, -15.376, -83.364, 50.813]
  Set speed (120.0 mm/s)
  MoveL 7875 to (497.72, 492.38, 15.8) mm, rotated rx 0 ry 90 rz 0 deg; joints [-11.351, -28.028, 112.026, -15.354, -83.348, 50.815]
  Set speed (30.0 mm/s)
  Call Extruder(0.070)
  MoveL 7876 to (499.42, 490.68, 15.8) mm, rotated rx 0 ry 90 rz 0 deg; joints [-11.163, -28.004, 111.864, -15.169, -83.21, 50.832]
  Set speed (120.0 mm/s)
  MoveL 7877 to (500.58, 490.68, 15.8) mm, rotated rx 0 ry 90 rz 0 deg; joints [-11.142, -27.982, 111.725, -15.151, -83.096, 50.861]
  Set speed (30.0 mm/s)
  Call Extruder(0.044)
  MoveL 7878 to (501.64, 491.74, 15.8) mm, rotated rx 0 ry 90 rz 0 deg; joints [-11.22, -27.958, 111.573, -15.234, -82.975, 50.903]
  Set speed (120.0 mm/s)
  MoveL 7879 to (502.48, 492.58, 15.8) mm, rotated rx 0 ry 90 rz 0 deg; joints [-11.282, -27.939, 111.452, -15.3, -82.878, 50.937]
  Set speed (30.0 mm/s)
  Call Extruder(0.281)
  MoveL 7880 to (509.32, 499.42, 15.8) mm, rotated rx 0 ry 90 rz 0 deg; joints [-11.777, -27.778, 110.462, -15.829, -82.097, 51.219]
  Set speed (120.0 mm/s)
  MoveL 7881 to (509.32, 500.58, 15.8) mm, rotated rx 0 ry 90 rz 0 deg; joints [-11.882, -27.773, 110.433, -15.935, -82.077, 51.238]
  Set speed (30.0 mm/s)
  Call Extruder(0.048)
  MoveL 7882 to (508.15, 501.74, 15.8) mm, rotated rx 0 ry 90 rz 0 deg; joints [-12.009, -27.791, 110.544, -16.06, -82.17, 51.228]
  MoveL 7883 to (508.03, 501.87, 15.8) mm, rotated rx 0 ry 90 rz 0 deg; joints [-12.023, -27.793, 110.556, -16.074, -82.18, 51.227]
  Set speed (120.0 mm/s)
  MoveL 7884 to (507.65, 497.03, 15.8) mm, rotated rx 0 ry 90 rz 0 deg; joints [-11.592, -27.821, 110.724, -15.634, -82.3, 51.136]
  Set speed (1000.0 mm/s)
  MoveL 7885 to (507.65, 494.43, 15.8) mm, rotated rx 0 ry 90 rz 0 deg; joints [-11.356, -27.832, 110.787, -15.394, -82.343, 51.094]
  Set speed (1000.0 mm/s)
  MoveL 7886 to (509.32, 490.68, 15.8) mm, rotated rx 0 ry 90 rz 0 deg; joints [-10.985, -27.813, 110.675, -15.023, -82.241, 51.074]
  Set speed (30.0 mm/s)
  Call Extruder(0.767)
  MoveL 7887 to (490.68, 509.32, 15.8) mm, rotated rx 0 ry 90 rz 0 deg; joints [-13.056, -28.089, 112.427, -17.058, -83.723, 50.887]
  MoveL 7888 to (490.56, 509.44, 15.8) mm, rotated rx 0 ry 90 rz 0 deg; joints [-13.07, -28.09, 112.438, -17.072, -83.733, 50.885]
  Set speed (120.0 mm/s)
  MoveL 7889 to (494.91, 492.37, 15.8) mm, rotated rx 0 ry 90 rz 0 deg; joints [-11.402, -28.079, 112.36, -15.397, -83.623, 50.744]
  Set speed (1000.0 mm/s)
  MoveL 7890 to (494.98, 492.3, 15.8) mm, rotated rx 0 ry 90 rz 0 deg; joints [-11.395, -28.078, 112.354, -15.39, -83.617, 50.745]
  Set speed (15.0 mm/s)
  Call Extruder(0.071)
  MoveL 7891 to (497.44, 492.3, 15.8) mm, rotated rx 0 ry 90 rz 0 deg; joints [-11.349, -28.034, 112.061, -15.351, -83.377, 50.807]
  Call Extruder(0.055)
  MoveL 7892 to (497.44, 490.4, 15.8) mm, rotated rx 0 ry 90 rz 0 deg; joints [-11.173, -28.041, 112.106, -15.173, -83.409, 50.779]
  Call Extruder(0.130)
  MoveL 7893 to (501.92, 490.4, 15.8) mm, rotated rx 0 ry 90 rz 0 deg; joints [-11.092, -27.958, 111.571, -15.105, -82.969, 50.889]
  Call Extruder(0.041)
  MoveL 7894 to (501.92, 491.81, 15.8) mm, rotated rx 0 ry 90 rz 0 deg; joints [-11.221, -27.953, 111.538, -15.236, -82.946, 50.911]
  Call Extruder(0.014)
  MoveL 7895 to (501.93, 492.3, 15.8) mm, rotated rx 0 ry 90 rz 0 deg; joints [-11.266, -27.951, 111.525, -15.282, -82.937, 50.919]
  Call Extruder(0.061)
  MoveL 7896 to (504.02, 492.3, 15.8) mm, rotated rx 0 ry 90 rz 0 deg; joints [-11.228, -27.911, 111.274, -15.251, -82.732, 50.97]
  Call Extruder(0.010)
  MoveL 7897 to (504.37, 492.3, 15.8) mm, rotated rx 0 ry 90 rz 0 deg; joints [-11.222, -27.904, 111.232, -15.245, -82.698, 50.979]
  Call Extruder(0.007)
  MoveL 7898 to (504.37, 491.95, 15.8) mm, rotated rx 0 ry 90 rz 0 deg; joints [-11.19, -27.906, 111.241, -15.213, -82.704, 50.974]
  Call Extruder(0.035)
  MoveL 7899 to (504.37, 490.75, 15.8) mm, rotated rx 0 ry 90 rz 0 deg; joints [-11.08, -27.91, 111.269, -15.101, -82.724, 50.955]
  Call Extruder(0.010)
  MoveL 7900 to (504.37, 490.4, 15.8) mm, rotated rx 0 ry 90 rz 0 deg; joints [-11.048, -27.912, 111.277, -15.069, -82.729, 50.949]
  Call Extruder(0.007)
  MoveL 7901 to (504.72, 490.4, 15.8) mm, rotated rx 0 ry 90 rz 0 deg; joints [-11.041, -27.905, 111.235, -15.064, -82.695, 50.958]
  Call Extruder(0.142)
  MoveL 7902 to (509.6, 490.4, 15.8) mm, rotated rx 0 ry 90 rz 0 deg; joints [-10.955, -27.809, 110.647, -14.993, -82.217, 51.076]
  Call Extruder(0.118)
  MoveL 7903 to (509.6, 494.46, 15.8) mm, rotated rx 0 ry 90 rz 0 deg; joints [-11.323, -27.793, 110.551, -15.368, -82.152, 51.143]
  Call Extruder(0.056)
  MoveL 7904 to (507.67, 494.46, 15.8) mm, rotated rx 0 ry 90 rz 0 deg; joints [-11.358, -27.831, 110.783, -15.396, -82.34, 51.095]
  Call Extruder(0.064)
  MoveL 7905 to (507.67, 496.65, 15.8) mm, rotated rx 0 ry 90 rz 0 deg; joints [-11.557, -27.822, 110.73, -15.598, -82.303, 51.131]
  Call Extruder(0.010)
  MoveL 7906 to (507.67, 497, 15.8) mm, rotated rx 0 ry 90 rz 0 deg; joints [-11.589, -27.821, 110.721, -15.631, -82.298, 51.137]
  Call Extruder(0.007)
  MoveL 7907 to (508.02, 497, 15.8) mm, rotated rx 0 ry 90 rz 0 deg; joints [-11.582, -27.814, 110.679, -15.625, -82.263, 51.145]
  Call Extruder(0.046)
  MoveL 7908 to (509.6, 497, 15.8) mm, rotated rx 0 ry 90 rz 0 deg; joints [-11.553, -27.782, 110.489, -15.602, -82.11, 51.185]
  Call Extruder(0.136)
  MoveL 7909 to (509.6, 501.68, 15.8) mm, rotated rx 0 ry 90 rz 0 deg; joints [-11.976, -27.762, 110.371, -16.032, -82.031, 51.264]
  Call Extruder(0.010)
  MoveL 7910 to (509.6, 502.03, 15.8) mm, rotated rx 0 ry 90 rz 0 deg; joints [-12.007, -27.761, 110.362, -16.064, -82.025, 51.27]
  Call Extruder(0.007)
  MoveL 7911 to (509.25, 502.03, 15.8) mm, rotated rx 0 ry 90 rz 0 deg; joints [-12.014, -27.768, 110.404, -16.069, -82.059, 51.261]
  Call Extruder(0.036)
  MoveL 7912 to (508.02, 502.02, 15.8) mm, rotated rx 0 ry 90 rz 0 deg; joints [-12.037, -27.793, 110.552, -16.088, -82.178, 51.23]
  Call Extruder(0.010)
  MoveL 7913 to (507.67, 502.02, 15.8) mm, rotated rx 0 ry 90 rz 0 deg; joints [-12.044, -27.8, 110.595, -16.094, -82.212, 51.221]
  Call Extruder(0.007)
  MoveL 7914 to (507.67, 502.37, 15.8) mm, rotated rx 0 ry 90 rz 0 deg; joints [-12.076, -27.798, 110.586, -16.126, -82.206, 51.227]
  Call Extruder(0.063)
  MoveL 7915 to (507.67, 504.54, 15.8) mm, rotated rx 0 ry 90 rz 0 deg; joints [-12.271, -27.789, 110.529, -16.325, -82.168, 51.264]
  Call Extruder(0.056)
  MoveL 7916 to (509.6, 504.54, 15.8) mm, rotated rx 0 ry 90 rz 0 deg; joints [-12.234, -27.75, 110.297, -16.295, -81.981, 51.314]
  Call Extruder(0.147)
  MoveL 7917 to (509.6, 509.6, 15.8) mm, rotated rx 0 ry 90 rz 0 deg; joints [-12.688, -27.727, 110.162, -16.758, -81.891, 51.403]
  Call Extruder(0.559)
  MoveL 7918 to (490.4, 509.6, 15.8) mm, rotated rx 0 ry 90 rz 0 deg; joints [-13.088, -28.092, 112.452, -17.09, -83.745, 50.883]
  MoveL 7919 to (490.4, 490.4, 15.8) mm, rotated rx 0 ry 90 rz 0 deg; joints [-11.303, -28.163, 112.942, -15.283, -84.101, 50.603]
  Call Extruder(0.134)
  MoveL 7920 to (494.99, 490.4, 15.8) mm, rotated rx 0 ry 90 rz 0 deg; joints [-11.218, -28.084, 112.398, -15.211, -83.649, 50.718]
  Call Extruder(0.041)
  MoveL 7921 to (494.99, 491.82, 15.8) mm, rotated rx 0 ry 90 rz 0 deg; joints [-11.35, -28.079, 112.364, -15.344, -83.625, 50.738]
  Call Extruder(0.014)
  MoveL 7922 to (494.98, 492.3, 15.8) mm, rotated rx 0 ry 90 rz 0 deg; joints [-11.395, -28.078, 112.354, -15.39, -83.617, 50.745]
  Set speed (120.0 mm/s)
  MoveL 7923 to (495.38, 492.3, 15.8) mm, rotated rx 0 ry 90 rz 0 deg; joints [-11.387, -28.071, 112.306, -15.383, -83.578, 50.755]
  Set speed (1000.0 mm/s)
  MoveL 7924 to (495.38, 493, 15.8) mm, rotated rx 0 ry 90 rz 0 deg; joints [-11.452, -28.068, 112.289, -15.449, -83.566, 50.765]
  Set speed (1000.0 mm/s)
  MoveL 7925 to (490.68, 490.68, 15.8) mm, rotated rx 0 ry 90 rz 0 deg; joints [-11.324, -28.158, 112.903, -15.305, -84.068, 50.613]
  Set speed (1000.0 mm/s)
  MoveL 7926 to (490.68, 490.68, 15.9) mm, rotated rx 0 ry 90 rz 0 deg; joints [-11.324, -28.168, 112.908, -15.305, -84.063, 50.615]
  Set speed (30.0 mm/s)
  Call Extruder(0.767)
  MoveL 7927 to (509.32, 509.32, 15.9) mm, rotated rx 0 ry 90 rz 0 deg; joints [-12.669, -27.744, 110.209, -16.737, -81.918, 51.393]
  MoveL 7928 to (509.44, 509.44, 15.9) mm, rotated rx 0 ry 90 rz 0 deg; joints [-12.677, -27.741, 110.191, -16.746, -81.904, 51.398]
  Set speed (120.0 mm/s)
  MoveL 7929 to (507.64, 504.63, 15.9) mm, rotated rx 0 ry 90 rz 0 deg; joints [-12.28, -27.8, 110.536, -16.333, -82.164, 51.266]
  Set speed (1000.0 mm/s)
  MoveL 7930 to (507.39, 502.51, 15.9) mm, rotated rx 0 ry 90 rz 0 deg; joints [-12.093, -27.814, 110.621, -16.143, -82.225, 51.223]
  Set speed (30.0 mm/s)
  Call Extruder(0.280)
  MoveL 7931 to (500.58, 509.32, 15.9) mm, rotated rx 0 ry 90 rz 0 deg; joints [-12.847, -27.918, 111.257, -16.883, -82.761, 51.159]
  Set speed (120.0 mm/s)
  MoveL 7932 to (499.42, 509.32, 15.9) mm, rotated rx 0 ry 90 rz 0 deg; joints [-12.872, -27.94, 111.395, -16.903, -82.873, 51.127]
  Set speed (30.0 mm/s)
  Call Extruder(0.360)
  MoveL 7933 to (490.68, 500.58, 15.9) mm, rotated rx 0 ry 90 rz 0 deg; joints [-12.247, -28.133, 112.664, -16.239, -83.885, 50.756]
  Set speed (120.0 mm/s)
  MoveL 7934 to (490.68, 499.42, 15.9) mm, rotated rx 0 ry 90 rz 0 deg; joints [-12.139, -28.137, 112.693, -16.13, -83.907, 50.739]
  Set speed (30.0 mm/s)
  Call Extruder(0.281)
  MoveL 7935 to (497.52, 492.58, 15.9) mm, rotated rx 0 ry 90 rz 0 deg; joints [-11.373, -28.042, 112.05, -15.376, -83.359, 50.814]
  Set speed (120.0 mm/s)
  MoveL 7936 to (497.66, 492.44, 15.9) mm, rotated rx 0 ry 90 rz 0 deg; joints [-11.357, -28.04, 112.037, -15.36, -83.347, 50.816]
  Set speed (30.0 mm/s)
  Call Extruder(0.072)
  MoveL 7937 to (499.42, 490.68, 15.9) mm, rotated rx 0 ry 90 rz 0 deg; joints [-11.163, -28.014, 111.869, -15.169, -83.205, 50.833]
  Set speed (120.0 mm/s)
  MoveL 7938 to (500.58, 490.68, 15.9) mm, rotated rx 0 ry 90 rz 0 deg; joints [-11.142, -27.993, 111.73, -15.151, -83.091, 50.862]
  Set speed (30.0 mm/s)
  Call Extruder(0.046)
  MoveL 7939 to (501.7, 491.81, 15.9) mm, rotated rx 0 ry 90 rz 0 deg; joints [-11.225, -27.968, 111.569, -15.239, -82.962, 50.907]
  Set speed (120.0 mm/s)
  MoveL 7940 to (502.48, 492.58, 15.9) mm, rotated rx 0 ry 90 rz 0 deg; joints [-11.282, -27.95, 111.457, -15.3, -82.873, 50.938]
  Set speed (30.0 mm/s)
  Call Extruder(0.281)
  MoveL 7941 to (509.32, 499.42, 15.9) mm, rotated rx 0 ry 90 rz 0 deg; joints [-11.777, -27.788, 110.467, -15.829, -82.091, 51.22]
  Set speed (120.0 mm/s)
  MoveL 7942 to (509.32, 500.58, 15.9) mm, rotated rx 0 ry 90 rz 0 deg; joints [-11.882, -27.783, 110.438, -15.935, -82.072, 51.24]
  Set speed (30.0 mm/s)
  Call Extruder(0.050)
  MoveL 7943 to (508.1, 501.8, 15.9) mm, rotated rx 0 ry 90 rz 0 deg; joints [-12.016, -27.803, 110.554, -16.067, -82.169, 51.229]
  MoveL 7944 to (507.97, 501.92, 15.9) mm, rotated rx 0 ry 90 rz 0 deg; joints [-12.029, -27.805, 110.566, -16.08, -82.179, 51.228]
  Set speed (120.0 mm/s)
  MoveL 7945 to (507.65, 496.97, 15.9) mm, rotated rx 0 ry 90 rz 0 deg; joints [-11.587, -27.832, 110.73, -15.628, -82.296, 51.137]
  Set speed (1000.0 mm/s)
  MoveL 7946 to (507.65, 494.37, 15.9) mm, rotated rx 0 ry 90 rz 0 deg; joints [-11.351, -27.843, 110.793, -15.389, -82.339, 51.094]
  Set speed (1000.0 mm/s)
  MoveL 7947 to (509.32, 490.68, 15.9) mm, rotated rx 0 ry 90 rz 0 deg; joints [-10.985, -27.824, 110.68, -15.023, -82.235, 51.076]
  Set speed (30.0 mm/s)
  Call Extruder(0.767)
  MoveL 7948 to (490.68, 509.32, 15.9) mm, rotated rx 0 ry 90 rz 0 deg; joints [-13.056, -28.099, 112.432, -17.059, -83.718, 50.888]
  MoveL 7949 to (490.56, 509.44, 15.9) mm, rotated rx 0 ry 90 rz 0 deg; joints [-13.07, -28.101, 112.443, -17.072, -83.728, 50.887]
  Set speed (120.0 mm/s)
  MoveL 7950 to (494.85, 492.37, 15.9) mm, rotated rx 0 ry 90 rz 0 deg; joints [-11.403, -28.09, 112.373, -15.398, -83.624, 50.744]
  Set speed (1000.0 mm/s)
  MoveL 7951 to (494.92, 492.3, 15.9) mm, rotated rx 0 ry 90 rz 0 deg; joints [-11.396, -28.089, 112.366, -15.391, -83.618, 50.745]
  Set speed (15.0 mm/s)
  Call Extruder(0.072)
  MoveL 7952 to (497.38, 492.3, 15.9) mm, rotated rx 0 ry 90 rz 0 deg; joints [-11.35, -28.045, 112.073, -15.352, -83.377, 50.807]
  Call Extruder(0.055)
  MoveL 7953 to (497.38, 490.4, 15.9) mm, rotated rx 0 ry 90 rz 0 deg; joints [-11.174, -28.052, 112.118, -15.174, -83.409, 50.779]
  Call Extruder(0.134)
  MoveL 7954 to (501.98, 490.4, 15.9) mm, rotated rx 0 ry 90 rz 0 deg; joints [-11.09, -27.968, 111.568, -15.104, -82.958, 50.892]
  Call Extruder(0.042)
  MoveL 7955 to (501.99, 491.85, 15.9) mm, rotated rx 0 ry 90 rz 0 deg; joints [-11.223, -27.962, 111.534, -15.239, -82.934, 50.915]
  Call Extruder(0.013)
  MoveL 7956 to (501.99, 492.3, 15.9) mm, rotated rx 0 ry 90 rz 0 deg; joints [-11.265, -27.96, 111.522, -15.281, -82.925, 50.922]
  Call Extruder(0.061)
  MoveL 7957 to (504.08, 492.3, 15.9) mm, rotated rx 0 ry 90 rz 0 deg; joints [-11.227, -27.92, 111.272, -15.25, -82.721, 50.973]
  Call Extruder(0.010)
  MoveL 7958 to (504.43, 492.3, 15.9) mm, rotated rx 0 ry 90 rz 0 deg; joints [-11.221, -27.914, 111.23, -15.245, -82.687, 50.982]
  Call Extruder(0.007)
  MoveL 7959 to (504.43, 491.95, 15.9) mm, rotated rx 0 ry 90 rz 0 deg; joints [-11.188, -27.915, 111.238, -15.212, -82.692, 50.977]
  Call Extruder(0.035)
  MoveL 7960 to (504.43, 490.75, 15.9) mm, rotated rx 0 ry 90 rz 0 deg; joints [-11.079, -27.92, 111.266, -15.101, -82.712, 50.958]
  Call Extruder(0.010)
  MoveL 7961 to (504.43, 490.4, 15.9) mm, rotated rx 0 ry 90 rz 0 deg; joints [-11.046, -27.921, 111.275, -15.068, -82.718, 50.952]
  Call Extruder(0.007)
  MoveL 7962 to (504.78, 490.4, 15.9) mm, rotated rx 0 ry 90 rz 0 deg; joints [-11.04, -27.914, 111.233, -15.063, -82.684, 50.961]
  Call Extruder(0.140)
  MoveL 7963 to (509.6, 490.4, 15.9) mm, rotated rx 0 ry 90 rz 0 deg; joints [-10.955, -27.819, 110.652, -14.994, -82.212, 51.078]
  Call Extruder(0.116)
  MoveL 7964 to (509.6, 494.4, 15.9) mm, rotated rx 0 ry 90 rz 0 deg; joints [-11.318, -27.803, 110.557, -15.363, -82.148, 51.143]
  Call Extruder(0.056)
  MoveL 7965 to (507.67, 494.4, 15.9) mm, rotated rx 0 ry 90 rz 0 deg; joints [-11.353, -27.842, 110.789, -15.391, -82.335, 51.096]
  Call Extruder(0.064)
  MoveL 7966 to (507.67, 496.59, 15.9) mm, rotated rx 0 ry 90 rz 0 deg; joints [-11.552, -27.833, 110.736, -15.593, -82.299, 51.131]
  Call Extruder(0.010)
  MoveL 7967 to (507.67, 496.94, 15.9) mm, rotated rx 0 ry 90 rz 0 deg; joints [-11.584, -27.832, 110.727, -15.625, -82.293, 51.137]
  Call Extruder(0.007)
  MoveL 7968 to (508.02, 496.94, 15.9) mm, rotated rx 0 ry 90 rz 0 deg; joints [-11.577, -27.825, 110.685, -15.62, -82.259, 51.146]
  Call Extruder(0.046)
  MoveL 7969 to (509.6, 496.94, 15.9) mm, rotated rx 0 ry 90 rz 0 deg; joints [-11.548, -27.793, 110.495, -15.597, -82.106, 51.185]
  Call Extruder(0.139)
  MoveL 7970 to (509.6, 501.73, 15.9) mm, rotated rx 0 ry 90 rz 0 deg; joints [-11.981, -27.773, 110.375, -16.037, -82.025, 51.267]
  Call Extruder(0.010)
  MoveL 7971 to (509.6, 502.08, 15.9) mm, rotated rx 0 ry 90 rz 0 deg; joints [-12.012, -27.771, 110.366, -16.069, -82.019, 51.273]
  Call Extruder(0.007)
  MoveL 7972 to (509.25, 502.08, 15.9) mm, rotated rx 0 ry 90 rz 0 deg; joints [-12.019, -27.778, 110.408, -16.075, -82.052, 51.264]
  Call Extruder(0.036)
  MoveL 7973 to (508.02, 502.08, 15.9) mm, rotated rx 0 ry 90 rz 0 deg; joints [-12.042, -27.803, 110.556, -16.093, -82.172, 51.232]
  Call Extruder(0.010)
  MoveL 7974 to (507.67, 502.08, 15.9) mm, rotated rx 0 ry 90 rz 0 deg; joints [-12.049, -27.81, 110.598, -16.099, -82.206, 51.223]
  Call Extruder(0.007)
  MoveL 7975 to (507.67, 502.43, 15.9) mm, rotated rx 0 ry 90 rz 0 deg; joints [-12.081, -27.809, 110.589, -16.131, -82.199, 51.229]
  Call Extruder(0.063)
  MoveL 7976 to (507.67, 504.6, 15.9) mm, rotated rx 0 ry 90 rz 0 deg; joints [-12.277, -27.799, 110.533, -16.33, -82.161, 51.266]
  Call Extruder(0.056)
  MoveL 7977 to (509.6, 504.6, 15.9) mm, rotated rx 0 ry 90 rz 0 deg; joints [-12.239, -27.76, 110.301, -16.3, -81.975, 51.316]
  Call Extruder(0.145)
  MoveL 7978 to (509.6, 509.6, 15.9) mm, rotated rx 0 ry 90 rz 0 deg; joints [-12.688, -27.737, 110.167, -16.758, -81.886, 51.405]
  Call Extruder(0.559)
  MoveL 7979 to (490.4, 509.6, 15.9) mm, rotated rx 0 ry 90 rz 0 deg; joints [-13.088, -28.103, 112.457, -17.09, -83.74, 50.885]
  MoveL 7980 to (490.4, 490.4, 15.9) mm, rotated rx 0 ry 90 rz 0 deg; joints [-11.303, -28.174, 112.948, -15.283, -84.095, 50.604]
  Call Extruder(0.132)
  MoveL 7981 to (494.93, 490.4, 15.9) mm, rotated rx 0 ry 90 rz 0 deg; joints [-11.219, -28.096, 112.41, -15.212, -83.65, 50.718]
  Call Extruder(0.042)
  MoveL 7982 to (494.93, 491.85, 15.9) mm, rotated rx 0 ry 90 rz 0 deg; joints [-11.354, -28.091, 112.376, -15.348, -83.625, 50.739]
  Call Extruder(0.013)
  MoveL 7983 to (494.92, 492.3, 15.9) mm, rotated rx 0 ry 90 rz 0 deg; joints [-11.396, -28.089, 112.366, -15.391, -83.618, 50.745]
  Set speed (120.0 mm/s)
  MoveL 7984 to (495.32, 492.3, 15.9) mm, rotated rx 0 ry 90 rz 0 deg; joints [-11.388, -28.082, 112.318, -15.384, -83.579, 50.755]
  Set speed (1000.0 mm/s)
  MoveL 7985 to (495.32, 493, 15.9) mm, rotated rx 0 ry 90 rz 0 deg; joints [-11.453, -28.08, 112.302, -15.45, -83.567, 50.765]
  Set speed (1000.0 mm/s)
  MoveL 7986 to (490.68, 490.68, 15.9) mm, rotated rx 0 ry 90 rz 0 deg; joints [-11.324, -28.168, 112.908, -15.305, -84.063, 50.615]
  Set speed (1000.0 mm/s)
  MoveL 7987 to (490.68, 490.68, 16) mm, rotated rx 0 ry 90 rz 0 deg; joints [-11.324, -28.179, 112.913, -15.305, -84.058, 50.616]
  Set speed (30.0 mm/s)
  Call Extruder(0.767)
  MoveL 7988 to (509.32, 509.32, 16) mm, rotated rx 0 ry 90 rz 0 deg; joints [-12.669, -27.755, 110.214, -16.737, -81.913, 51.394]
  MoveL 7989 to (509.44, 509.44, 16) mm, rotated rx 0 ry 90 rz 0 deg; joints [-12.677, -27.752, 110.196, -16.746, -81.898, 51.4]
  Set speed (120.0 mm/s)
  MoveL 7990 to (507.64, 504.68, 16) mm, rotated rx 0 ry 90 rz 0 deg; joints [-12.285, -27.81, 110.539, -16.339, -82.157, 51.269]
  Set speed (1000.0 mm/s)
  MoveL 7991 to (507.39, 502.51, 16) mm, rotated rx 0 ry 90 rz 0 deg; joints [-12.093, -27.825, 110.626, -16.143, -82.22, 51.225]
  Set speed (30.0 mm/s)
  Call Extruder(0.280)
  MoveL 7992 to (500.58, 509.32, 16) mm, rotated rx 0 ry 90 rz 0 deg; joints [-12.847, -27.929, 111.262, -16.883, -82.756, 51.16]
  Set speed (120.0 mm/s)
  MoveL 7993 to (499.42, 509.32, 16) mm, rotated rx 0 ry 90 rz 0 deg; joints [-12.872, -27.951, 111.4, -16.903, -82.868, 51.129]
  Set speed (30.0 mm/s)
  Call Extruder(0.360)
  MoveL 7994 to (490.68, 500.58, 16) mm, rotated rx 0 ry 90 rz 0 deg; joints [-12.247, -28.144, 112.669, -16.239, -83.88, 50.757]
  Set speed (120.0 mm/s)
  MoveL 7995 to (490.68, 499.42, 16) mm, rotated rx 0 ry 90 rz 0 deg; joints [-12.139, -28.148, 112.698, -16.13, -83.901, 50.74]
  Set speed (30.0 mm/s)
  Call Extruder(0.281)
  MoveL 7996 to (497.51, 492.59, 16) mm, rotated rx 0 ry 90 rz 0 deg; joints [-11.374, -28.053, 112.056, -15.377, -83.354, 50.816]
  Set speed (120.0 mm/s)
  MoveL 7997 to (497.59, 492.51, 16) mm, rotated rx 0 ry 90 rz 0 deg; joints [-11.365, -28.052, 112.049, -15.368, -83.348, 50.816]
  Set speed (30.0 mm/s)
  Call Extruder(0.075)
  MoveL 7998 to (499.42, 490.68, 16) mm, rotated rx 0 ry 90 rz 0 deg; joints [-11.163, -28.025, 111.874, -15.169, -83.199, 50.835]
  Set speed (120.0 mm/s)
  MoveL 7999 to (500.58, 490.68, 16) mm, rotated rx 0 ry 90 rz 0 deg; joints [-11.141, -28.003, 111.735, -15.152, -83.086, 50.863]
  Set speed (30.0 mm/s)
  Call Extruder(0.049)
  MoveL 8000 to (501.77, 491.87, 16) mm, rotated rx 0 ry 90 rz 0 deg; joints [-11.229, -27.977, 111.565, -15.245, -82.949, 50.911]
  Set speed (120.0 mm/s)
  MoveL 8001 to (502.47, 492.57, 16) mm, rotated rx 0 ry 90 rz 0 deg; joints [-11.28, -27.961, 111.465, -15.299, -82.87, 50.939]
  Set speed (30.0 mm/s)
  Call Extruder(0.282)
  MoveL 8002 to (509.31, 499.41, 16) mm, rotated rx 0 ry 90 rz 0 deg; joints [-11.777, -27.799, 110.474, -15.828, -82.087, 51.221]
  Set speed (120.0 mm/s)
  MoveL 8003 to (509.31, 500.58, 16) mm, rotated rx 0 ry 90 rz 0 deg; joints [-11.882, -27.794, 110.444, -15.936, -82.067, 51.241]
  Set speed (30.0 mm/s)
  Call Extruder(0.052)
  MoveL 8004 to (508.04, 501.86, 16) mm, rotated rx 0 ry 90 rz 0 deg; joints [-12.022, -27.814, 110.565, -16.073, -82.169, 51.23]
  MoveL 8005 to (507.92, 501.98, 16) mm, rotated rx 0 ry 90 rz 0 deg; joints [-12.035, -27.816, 110.576, -16.086, -82.178, 51.229]
  Set speed (120.0 mm/s)
  MoveL 8006 to (507.65, 496.9, 16) mm, rotated rx 0 ry 90 rz 0 deg; joints [-11.58, -27.843, 110.737, -15.622, -82.291, 51.137]
  Set speed (1000.0 mm/s)
  MoveL 8007 to (507.65, 494.32, 16) mm, rotated rx 0 ry 90 rz 0 deg; joints [-11.346, -27.853, 110.8, -15.384, -82.334, 51.095]
  Set speed (1000.0 mm/s)
  MoveL 8008 to (509.32, 490.68, 16) mm, rotated rx 0 ry 90 rz 0 deg; joints [-10.985, -27.834, 110.685, -15.024, -82.23, 51.077]
  Set speed (30.0 mm/s)
  Call Extruder(0.767)
  MoveL 8009 to (490.68, 509.32, 16) mm, rotated rx 0 ry 90 rz 0 deg; joints [-13.056, -28.11, 112.437, -17.059, -83.713, 50.89]
  MoveL 8010 to (490.56, 509.44, 16) mm, rotated rx 0 ry 90 rz 0 deg; joints [-13.07, -28.111, 112.448, -17.073, -83.722, 50.888]
  Set speed (120.0 mm/s)
  MoveL 8011 to (504.57, 492.38, 16) mm, rotated rx 0 ry 90 rz 0 deg; joints [-11.225, -27.921, 111.217, -15.25, -82.667, 50.988]
  Set speed (1000.0 mm/s)
  MoveL 8012 to (504.5, 492.31, 16) mm, rotated rx 0 ry 90 rz 0 deg; joints [-11.22, -27.923, 111.227, -15.244, -82.675, 50.985]
  Set speed (15.0 mm/s)
  Call Extruder(0.010)
  MoveL 8013 to (504.5, 491.95, 16) mm, rotated rx 0 ry 90 rz 0 deg; joints [-11.188, -27.924, 111.235, -15.212, -82.681, 50.98]
  Call Extruder(0.000)
  MoveL 8014 to (504.5, 491.95, 16) mm, rotated rx 0 ry 90 rz 0 deg; joints [-11.187, -27.924, 111.235, -15.212, -82.681, 50.98]
  Call Extruder(0.035)
  MoveL 8015 to (504.5, 490.75, 16) mm, rotated rx 0 ry 90 rz 0 deg; joints [-11.077, -27.929, 111.264, -15.1, -82.701, 50.961]
  Call Extruder(0.010)
  MoveL 8016 to (504.5, 490.4, 16) mm, rotated rx 0 ry 90 rz 0 deg; joints [-11.045, -27.93, 111.272, -15.067, -82.706, 50.955]
  Call Extruder(0.007)
  MoveL 8017 to (504.85, 490.4, 16) mm, rotated rx 0 ry 90 rz 0 deg; joints [-11.039, -27.923, 111.23, -15.062, -82.672, 50.964]
  Call Extruder(0.138)
  MoveL 8018 to (509.6, 490.4, 16) mm, rotated rx 0 ry 90 rz 0 deg; joints [-10.955, -27.83, 110.657, -14.994, -82.207, 51.079]
  Call Extruder(0.114)
  MoveL 8019 to (509.6, 494.33, 16) mm, rotated rx 0 ry 90 rz 0 deg; joints [-11.311, -27.814, 110.564, -15.356, -82.144, 51.143]
  Call Extruder(0.056)
  MoveL 8020 to (507.67, 494.35, 16) mm, rotated rx 0 ry 90 rz 0 deg; joints [-11.348, -27.853, 110.796, -15.386, -82.331, 51.096]
  Call Extruder(0.074)
  MoveL 8021 to (507.67, 496.87, 16) mm, rotated rx 0 ry 90 rz 0 deg; joints [-11.577, -27.843, 110.734, -15.619, -82.289, 51.138]
  Call Extruder(0.056)
  MoveL 8022 to (509.59, 496.88, 16) mm, rotated rx 0 ry 90 rz 0 deg; joints [-11.543, -27.804, 110.503, -15.591, -82.103, 51.186]
  Call Extruder(0.143)
  MoveL 8023 to (509.6, 501.79, 16) mm, rotated rx 0 ry 90 rz 0 deg; joints [-11.986, -27.783, 110.379, -16.042, -82.019, 51.269]
  Call Extruder(0.010)
  MoveL 8024 to (509.6, 502.14, 16) mm, rotated rx 0 ry 90 rz 0 deg; joints [-12.017, -27.781, 110.37, -16.075, -82.012, 51.275]
  Call Extruder(0.007)
  MoveL 8025 to (509.25, 502.14, 16) mm, rotated rx 0 ry 90 rz 0 deg; joints [-12.024, -27.789, 110.412, -16.08, -82.046, 51.266]
  Call Extruder(0.036)
  MoveL 8026 to (508.02, 502.14, 16) mm, rotated rx 0 ry 90 rz 0 deg; joints [-12.047, -27.813, 110.56, -16.099, -82.165, 51.235]
  Call Extruder(0.010)
  MoveL 8027 to (507.67, 502.14, 16) mm, rotated rx 0 ry 90 rz 0 deg; joints [-12.054, -27.82, 110.602, -16.104, -82.199, 51.226]
  Call Extruder(0.007)
  MoveL 8028 to (507.67, 502.49, 16) mm, rotated rx 0 ry 90 rz 0 deg; joints [-12.086, -27.819, 110.593, -16.137, -82.193, 51.232]
  Call Extruder(0.063)
  MoveL 8029 to (507.67, 504.66, 16) mm, rotated rx 0 ry 90 rz 0 deg; joints [-12.282, -27.81, 110.537, -16.336, -82.155, 51.269]
  Call Extruder(0.056)
  MoveL 8030 to (509.6, 504.66, 16) mm, rotated rx 0 ry 90 rz 0 deg; joints [-12.244, -27.77, 110.304, -16.306, -81.969, 51.319]
  Call Extruder(0.144)
  MoveL 8031 to (509.6, 509.6, 16) mm, rotated rx 0 ry 90 rz 0 deg; joints [-12.688, -27.748, 110.173, -16.758, -81.88, 51.407]
  Call Extruder(0.559)
  MoveL 8032 to (490.4, 509.6, 16) mm, rotated rx 0 ry 90 rz 0 deg; joints [-13.088, -28.114, 112.462, -17.09, -83.734, 50.887]
  MoveL 8033 to (490.4, 490.4, 16) mm, rotated rx 0 ry 90 rz 0 deg; joints [-11.303, -28.185, 112.953, -15.283, -84.09, 50.605]
  Call Extruder(0.130)
  MoveL 8034 to (494.88, 490.4, 16) mm, rotated rx 0 ry 90 rz 0 deg; joints [-11.22, -28.108, 112.422, -15.213, -83.65, 50.718]
  Call Extruder(0.055)
  MoveL 8035 to (494.88, 492.29, 16) mm, rotated rx 0 ry 90 rz 0 deg; joints [-11.395, -28.101, 112.377, -15.39, -83.618, 50.745]
  Call Extruder(0.061)
  MoveL 8036 to (496.96, 492.3, 16) mm, rotated rx 0 ry 90 rz 0 deg; joints [-11.358, -28.064, 112.128, -15.359, -83.413, 50.798]
  Call Extruder(0.010)
  MoveL 8037 to (497.31, 492.31, 16) mm, rotated rx 0 ry 90 rz 0 deg; joints [-11.351, -28.057, 112.086, -15.354, -83.378, 50.806]
  Call Extruder(0.007)
  MoveL 8038 to (497.31, 491.95, 16) mm, rotated rx 0 ry 90 rz 0 deg; joints [-11.319, -28.059, 112.095, -15.321, -83.384, 50.801]
  Call Extruder(0.045)
  MoveL 8039 to (497.33, 490.4, 16) mm, rotated rx 0 ry 90 rz 0 deg; joints [-11.175, -28.064, 112.13, -15.175, -83.409, 50.779]
  Call Extruder(0.137)
  MoveL 8040 to (502.05, 490.4, 16) mm, rotated rx 0 ry 90 rz 0 deg; joints [-11.089, -27.977, 111.566, -15.104, -82.946, 50.895]
  Call Extruder(0.055)
  MoveL 8041 to (502.05, 492.28, 16) mm, rotated rx 0 ry 90 rz 0 deg; joints [-11.262, -27.97, 111.521, -15.279, -82.915, 50.924]
  Call Extruder(0.061)
  MoveL 8042 to (504.15, 492.3, 16) mm, rotated rx 0 ry 90 rz 0 deg; joints [-11.226, -27.93, 111.269, -15.249, -82.71, 50.976]
  Call Extruder(0.000)
  MoveL 8043 to (504.15, 492.3, 16) mm, rotated rx 0 ry 90 rz 0 deg; joints [-11.226, -27.93, 111.269, -15.249, -82.71, 50.976]
  Call Extruder(0.007)
  MoveL 8044 to (504.5, 492.31, 16) mm, rotated rx 0 ry 90 rz 0 deg; joints [-11.22, -27.923, 111.227, -15.244, -82.675, 50.985]
  Set speed (120.0 mm/s)
  MoveL 8045 to (504.5, 491.95, 16) mm, rotated rx 0 ry 90 rz 0 deg; joints [-11.188, -27.924, 111.235, -15.212, -82.681, 50.98]
  Set speed (1000.0 mm/s)
  MoveL 8046 to (504.5, 491.95, 16) mm, rotated rx 0 ry 90 rz 0 deg; joints [-11.187, -27.924, 111.235, -15.212, -82.681, 50.98]
  Set speed (1000.0 mm/s)
  MoveL 8047 to (504.5, 491.91, 16) mm, rotated rx 0 ry 90 rz 0 deg; joints [-11.183, -27.925, 111.236, -15.207, -82.682, 50.979]
  Set speed (1000.0 mm/s)
  MoveL 8048 to (505.2, 491.91, 16) mm, rotated rx 0 ry 90 rz 0 deg; joints [-11.17, -27.911, 111.152, -15.197, -82.613, 50.996]
  Set speed (1000.0 mm/s)
  MoveL 8049 to (494.85, 492.32, 16) mm, rotated rx 0 ry 90 rz 0 deg; joints [-11.398, -28.101, 112.379, -15.393, -83.62, 50.745]
  Set speed (1000.0 mm/s)
  MoveL 8050 to (490.68, 490.68, 16) mm, rotated rx 0 ry 90 rz 0 deg; joints [-11.324, -28.179, 112.913, -15.305, -84.058, 50.616]
  Set speed (1000.0 mm/s)
  MoveL 8051 to (490.68, 490.68, 16.1) mm, rotated rx 0 ry 90 rz 0 deg; joints [-11.324, -28.19, 112.918, -15.306, -84.052, 50.618]
  Set speed (30.0 mm/s)
  Call Extruder(0.767)
  MoveL 8052 to (509.32, 509.32, 16.1) mm, rotated rx 0 ry 90 rz 0 deg; joints [-12.669, -27.765, 110.219, -16.737, -81.907, 51.396]
  MoveL 8053 to (509.44, 509.44, 16.1) mm, rotated rx 0 ry 90 rz 0 deg; joints [-12.677, -27.762, 110.201, -16.746, -81.893, 51.401]
  Set speed (120.0 mm/s)
  MoveL 8054 to (507.64, 504.74, 16.1) mm, rotated rx 0 ry 90 rz 0 deg; joints [-12.29, -27.82, 110.543, -16.344, -82.151, 51.271]
  Set speed (1000.0 mm/s)
  MoveL 8055 to (507.39, 502.51, 16.1) mm, rotated rx 0 ry 90 rz 0 deg; joints [-12.093, -27.835, 110.631, -16.143, -82.215, 51.226]
  Set speed (30.0 mm/s)
  Call Extruder(0.280)
  MoveL 8056 to (500.58, 509.32, 16.1) mm, rotated rx 0 ry 90 rz 0 deg; joints [-12.847, -27.939, 111.267, -16.883, -82.751, 51.162]
  Set speed (120.0 mm/s)
  MoveL 8057 to (499.42, 509.32, 16.1) mm, rotated rx 0 ry 90 rz 0 deg; joints [-12.872, -27.961, 111.405, -16.903, -82.863, 51.131]
  Set speed (30.0 mm/s)
  Call Extruder(0.360)
  MoveL 8058 to (490.68, 500.58, 16.1) mm, rotated rx 0 ry 90 rz 0 deg; joints [-12.247, -28.154, 112.674, -16.239, -83.875, 50.759]
  Set speed (120.0 mm/s)
  MoveL 8059 to (490.68, 499.42, 16.1) mm, rotated rx 0 ry 90 rz 0 deg; joints [-12.139, -28.159, 112.704, -16.13, -83.896, 50.742]
  Set speed (30.0 mm/s)
  MoveL 8060 to (499.42, 490.68, 16.1) mm, rotated rx 0 ry 90 rz 0 deg; joints [-11.163, -28.035, 111.879, -15.169, -83.194, 50.836]
  Set speed (120.0 mm/s)
  MoveL 8061 to (500.58, 490.68, 16.1) mm, rotated rx 0 ry 90 rz 0 deg; joints [-11.141, -28.014, 111.74, -15.152, -83.08, 50.865]
  Set speed (30.0 mm/s)
  Call Extruder(0.047)
  MoveL 8062 to (501.73, 491.83, 16.1) mm, rotated rx 0 ry 90 rz 0 deg; joints [-11.226, -27.988, 111.576, -15.241, -82.949, 50.911]
  Set speed (120.0 mm/s)
  MoveL 8063 to (502.08, 492.18, 16.1) mm, rotated rx 0 ry 90 rz 0 deg; joints [-11.252, -27.98, 111.525, -15.269, -82.908, 50.925]
  Set speed (30.0 mm/s)
  Call Extruder(0.298)
  MoveL 8064 to (509.32, 499.42, 16.1) mm, rotated rx 0 ry 90 rz 0 deg; joints [-11.777, -27.809, 110.478, -15.829, -82.081, 51.223]
  Set speed (120.0 mm/s)
  MoveL 8065 to (509.32, 500.58, 16.1) mm, rotated rx 0 ry 90 rz 0 deg; joints [-11.882, -27.804, 110.448, -15.936, -82.061, 51.243]
  Set speed (30.0 mm/s)
  Call Extruder(0.055)
  MoveL 8066 to (507.99, 501.91, 16.1) mm, rotated rx 0 ry 90 rz 0 deg; joints [-12.028, -27.826, 110.575, -16.079, -82.168, 51.231]
  MoveL 8067 to (507.86, 502.04, 16.1) mm, rotated rx 0 ry 90 rz 0 deg; joints [-12.041, -27.828, 110.587, -16.092, -82.177, 51.23]
  Set speed (120.0 mm/s)
  MoveL 8068 to (509.32, 490.68, 16.1) mm, rotated rx 0 ry 90 rz 0 deg; joints [-10.985, -27.845, 110.69, -15.024, -82.225, 51.078]
  Set speed (30.0 mm/s)
  Call Extruder(0.767)
  MoveL 8069 to (490.68, 509.32, 16.1) mm, rotated rx 0 ry 90 rz 0 deg; joints [-13.056, -28.12, 112.442, -17.059, -83.708, 50.891]
  MoveL 8070 to (490.56, 509.44, 16.1) mm, rotated rx 0 ry 90 rz 0 deg; joints [-13.07, -28.122, 112.453, -17.073, -83.717, 50.89]
  Set speed (120.0 mm/s)
  MoveL 8071 to (507.6, 502.12, 16.1) mm, rotated rx 0 ry 90 rz 0 deg; joints [-12.054, -27.832, 110.616, -16.104, -82.201, 51.225]
  Set speed (1000.0 mm/s)
  MoveL 8072 to (507.67, 502.19, 16.1) mm, rotated rx 0 ry 90 rz 0 deg; joints [-12.059, -27.831, 110.606, -16.11, -82.193, 51.228]
  Set speed (15.0 mm/s)
  Call Extruder(0.010)
  MoveL 8073 to (507.67, 502.54, 16.1) mm, rotated rx 0 ry 90 rz 0 deg; joints [-12.091, -27.829, 110.597, -16.142, -82.187, 51.234]
  Call Extruder(0.063)
  MoveL 8074 to (507.67, 504.71, 16.1) mm, rotated rx 0 ry 90 rz 0 deg; joints [-12.287, -27.82, 110.54, -16.341, -82.149, 51.271]
  Call Extruder(0.056)
  MoveL 8075 to (509.59, 504.71, 16.1) mm, rotated rx 0 ry 90 rz 0 deg; joints [-12.249, -27.781, 110.309, -16.311, -81.963, 51.321]
  Call Extruder(0.132)
  MoveL 8076 to (509.6, 509.25, 16.1) mm, rotated rx 0 ry 90 rz 0 deg; joints [-12.657, -27.76, 110.187, -16.726, -81.882, 51.402]
  Call Extruder(0.010)
  MoveL 8077 to (509.6, 509.6, 16.1) mm, rotated rx 0 ry 90 rz 0 deg; joints [-12.688, -27.758, 110.178, -16.758, -81.875, 51.408]
  Call Extruder(0.007)
  MoveL 8078 to (509.25, 509.6, 16.1) mm, rotated rx 0 ry 90 rz 0 deg; joints [-12.695, -27.765, 110.22, -16.764, -81.909, 51.399]
  Call Extruder(0.549)
  MoveL 8079 to (490.4, 509.6, 16.1) mm, rotated rx 0 ry 90 rz 0 deg; joints [-13.088, -28.124, 112.467, -17.09, -83.729, 50.888]
  Call Extruder(0.559)
  MoveL 8080 to (490.4, 490.4, 16.1) mm, rotated rx 0 ry 90 rz 0 deg; joints [-11.303, -28.195, 112.958, -15.284, -84.085, 50.607]
  MoveL 8081 to (509.6, 490.4, 16.1) mm, rotated rx 0 ry 90 rz 0 deg; joints [-10.955, -27.84, 110.663, -14.994, -82.202, 51.081]
  Call Extruder(0.333)
  MoveL 8082 to (509.6, 501.85, 16.1) mm, rotated rx 0 ry 90 rz 0 deg; joints [-11.991, -27.793, 110.382, -16.048, -82.012, 51.272]
  Call Extruder(0.010)
  MoveL 8083 to (509.6, 502.2, 16.1) mm, rotated rx 0 ry 90 rz 0 deg; joints [-12.022, -27.792, 110.373, -16.08, -82.006, 51.278]
  Call Extruder(0.007)
  MoveL 8084 to (509.25, 502.19, 16.1) mm, rotated rx 0 ry 90 rz 0 deg; joints [-12.029, -27.799, 110.415, -16.085, -82.04, 51.269]
  Call Extruder(0.036)
  MoveL 8085 to (508.02, 502.19, 16.1) mm, rotated rx 0 ry 90 rz 0 deg; joints [-12.052, -27.824, 110.563, -16.104, -82.159, 51.237]
  Call Extruder(0.007)
  MoveL 8086 to (507.67, 502.19, 16.1) mm, rotated rx 0 ry 90 rz 0 deg; joints [-12.059, -27.831, 110.606, -16.11, -82.193, 51.228]
  Set speed (120.0 mm/s)
  MoveL 8087 to (507.67, 502.54, 16.1) mm, rotated rx 0 ry 90 rz 0 deg; joints [-12.091, -27.829, 110.597, -16.142, -82.187, 51.234]
  Set speed (1000.0 mm/s)
  MoveL 8088 to (507.67, 502.59, 16.1) mm, rotated rx 0 ry 90 rz 0 deg; joints [-12.095, -27.829, 110.595, -16.146, -82.186, 51.235]
  Set speed (1000.0 mm/s)
  MoveL 8089 to (507.57, 502.59, 16.1) mm, rotated rx 0 ry 90 rz 0 deg; joints [-12.097, -27.831, 110.607, -16.148, -82.196, 51.232]
  Set speed (1000.0 mm/s)
  MoveL 8090 to (507.71, 497.25, 16.1) mm, rotated rx 0 ry 90 rz 0 deg; joints [-11.611, -27.851, 110.725, -15.654, -82.274, 51.146]
  Set speed (15.0 mm/s)
  Call Extruder(0.051)
  MoveL 8091 to (507.71, 495.51, 16.1) mm, rotated rx 0 ry 90 rz 0 deg; joints [-11.453, -27.858, 110.768, -15.493, -82.303, 51.118]
  Call Extruder(0.033)
  MoveL 8092 to (507.72, 494.39, 16.1) mm, rotated rx 0 ry 90 rz 0 deg; joints [-11.351, -27.862, 110.795, -15.389, -82.321, 51.099]
  Call Extruder(0.035)
  MoveL 8093 to (508.91, 494.38, 16.1) mm, rotated rx 0 ry 90 rz 0 deg; joints [-11.328, -27.838, 110.651, -15.371, -82.205, 51.129]
  Call Extruder(0.084)
  MoveL 8094 to (508.91, 497.25, 16.1) mm, rotated rx 0 ry 90 rz 0 deg; joints [-11.589, -27.827, 110.581, -15.636, -82.157, 51.176]
  Call Extruder(0.035)
  MoveL 8095 to (507.71, 497.25, 16.1) mm, rotated rx 0 ry 90 rz 0 deg; joints [-11.611, -27.851, 110.725, -15.654, -82.274, 51.146]
  Set speed (120.0 mm/s)
  MoveL 8096 to (508.59, 496.71, 16.1) mm, rotated rx 0 ry 90 rz 0 deg; joints [-11.546, -27.835, 110.632, -15.591, -82.197, 51.159]
  Set speed (15.0 mm/s)
  Call Extruder(0.023)
  MoveL 8097 to (508.03, 496.15, 16.1) mm, rotated rx 0 ry 90 rz 0 deg; joints [-11.505, -27.849, 110.715, -15.547, -82.262, 51.136]
  Set speed (120.0 mm/s)
  MoveL 8098 to (508.59, 495.72, 16.1) mm, rotated rx 0 ry 90 rz 0 deg; joints [-11.456, -27.839, 110.657, -15.5, -82.214, 51.143]
  Set speed (15.0 mm/s)
  Call Extruder(0.023)
  MoveL 8099 to (508.03, 495.16, 16.1) mm, rotated rx 0 ry 90 rz 0 deg; joints [-11.415, -27.853, 110.739, -15.456, -82.278, 51.12]
  Set speed (120.0 mm/s)
  MoveL 8100 to (504.46, 492.27, 16.1) mm, rotated rx 0 ry 90 rz 0 deg; joints [-11.217, -27.934, 111.238, -15.242, -82.674, 50.985]
  Set speed (15.0 mm/s)
  Call Extruder(0.016)
  MoveL 8101 to (503.92, 492.26, 16.1) mm, rotated rx 0 ry 90 rz 0 deg; joints [-11.226, -27.945, 111.302, -15.249, -82.727, 50.972]
  Call Extruder(0.066)
  MoveL 8102 to (501.65, 492.26, 16.1) mm, rotated rx 0 ry 90 rz 0 deg; joints [-11.268, -27.988, 111.575, -15.283, -82.949, 50.915]
  Call Extruder(0.034)
  MoveL 8103 to (501.65, 491.09, 16.1) mm, rotated rx 0 ry 90 rz 0 deg; joints [-11.16, -27.992, 111.603, -15.174, -82.969, 50.897]
  Call Extruder(0.082)
  MoveL 8104 to (504.46, 491.09, 16.1) mm, rotated rx 0 ry 90 rz 0 deg; joints [-11.109, -27.939, 111.266, -15.132, -82.694, 50.967]
  Call Extruder(0.034)
  MoveL 8105 to (504.46, 492.27, 16.1) mm, rotated rx 0 ry 90 rz 0 deg; joints [-11.217, -27.934, 111.238, -15.242, -82.674, 50.985]
  Set speed (120.0 mm/s)
  MoveL 8106 to (503.82, 491.95, 16.1) mm, rotated rx 0 ry 90 rz 0 deg; joints [-11.199, -27.948, 111.321, -15.221, -82.742, 50.964]
  Set speed (15.0 mm/s)
  Call Extruder(0.022)
  MoveL 8107 to (503.28, 491.41, 16.1) mm, rotated rx 0 ry 90 rz 0 deg; joints [-11.159, -27.96, 111.399, -15.179, -82.803, 50.943]
  Set speed (120.0 mm/s)
  MoveL 8108 to (502.84, 491.95, 16.1) mm, rotated rx 0 ry 90 rz 0 deg; joints [-11.217, -27.967, 111.44, -15.236, -82.838, 50.94]
  Set speed (15.0 mm/s)
  MoveL 8109 to (502.29, 491.4, 16.1) mm, rotated rx 0 ry 90 rz 0 deg; joints [-11.177, -27.979, 111.518, -15.194, -82.9, 50.918]
  Set speed (120.0 mm/s)
  MoveL 8110 to (497.68, 491.09, 16.1) mm, rotated rx 0 ry 90 rz 0 deg; joints [-11.232, -28.066, 112.076, -15.234, -83.357, 50.799]
  Set speed (15.0 mm/s)
  Call Extruder(0.034)
  MoveL 8111 to (497.68, 492.26, 16.1) mm, rotated rx 0 ry 90 rz 0 deg; joints [-11.341, -28.061, 112.049, -15.344, -83.338, 50.816]
  Call Extruder(0.079)
  MoveL 8112 to (494.97, 492.26, 16.1) mm, rotated rx 0 ry 90 rz 0 deg; joints [-11.391, -28.11, 112.371, -15.386, -83.603, 50.748]
  Call Extruder(0.000)
  MoveL 8113 to (494.97, 492.25, 16.1) mm, rotated rx 0 ry 90 rz 0 deg; joints [-11.39, -28.11, 112.371, -15.386, -83.603, 50.748]
  Call Extruder(0.002)
  MoveL 8114 to (494.92, 492.25, 16.1) mm, rotated rx 0 ry 90 rz 0 deg; joints [-11.391, -28.111, 112.378, -15.386, -83.609, 50.747]
  Call Extruder(0.034)
  MoveL 8115 to (494.92, 491.09, 16.1) mm, rotated rx 0 ry 90 rz 0 deg; joints [-11.283, -28.115, 112.406, -15.277, -83.629, 50.73]
  Call Extruder(0.081)
  MoveL 8116 to (497.68, 491.09, 16.1) mm, rotated rx 0 ry 90 rz 0 deg; joints [-11.232, -28.066, 112.076, -15.234, -83.357, 50.799]
  Set speed (120.0 mm/s)
  MoveL 8117 to (496.89, 491.95, 16.1) mm, rotated rx 0 ry 90 rz 0 deg; joints [-11.326, -28.077, 112.15, -15.327, -83.42, 50.792]
  Set speed (15.0 mm/s)
  Call Extruder(0.022)
  MoveL 8118 to (496.35, 491.4, 16.1) mm, rotated rx 0 ry 90 rz 0 deg; joints [-11.286, -28.088, 112.227, -15.284, -83.482, 50.771]
  Set speed (120.0 mm/s)
  MoveL 8119 to (495.91, 491.95, 16.1) mm, rotated rx 0 ry 90 rz 0 deg; joints [-11.344, -28.095, 112.268, -15.342, -83.517, 50.767]
  Set speed (15.0 mm/s)
  Call Extruder(0.022)
  MoveL 8120 to (495.36, 491.4, 16.1) mm, rotated rx 0 ry 90 rz 0 deg; joints [-11.304, -28.106, 112.345, -15.3, -83.58, 50.746]
  Set speed (120.0 mm/s)
  MoveL 8121 to (490.68, 490.68, 16.1) mm, rotated rx 0 ry 90 rz 0 deg; joints [-11.324, -28.19, 112.918, -15.306, -84.052, 50.618]
  Set speed (1000.0 mm/s)
  MoveL 8122 to (490.68, 490.68, 16.2) mm, rotated rx 0 ry 90 rz 0 deg; joints [-11.324, -28.2, 112.923, -15.306, -84.047, 50.619]
  Set speed (30.0 mm/s)
  Call Extruder(0.767)
  MoveL 8123 to (509.32, 509.32, 16.2) mm, rotated rx 0 ry 90 rz 0 deg; joints [-12.669, -27.776, 110.224, -16.737, -81.902, 51.397]
  MoveL 8124 to (509.44, 509.44, 16.2) mm, rotated rx 0 ry 90 rz 0 deg; joints [-12.677, -27.773, 110.206, -16.747, -81.888, 51.403]
  Set speed (120.0 mm/s)
  MoveL 8125 to (507.79, 502.11, 16.2) mm, rotated rx 0 ry 90 rz 0 deg; joints [-12.049, -27.839, 110.599, -16.1, -82.178, 51.231]
  Set speed (30.0 mm/s)
  Call Extruder(0.297)
  MoveL 8126 to (500.58, 509.32, 16.2) mm, rotated rx 0 ry 90 rz 0 deg; joints [-12.847, -27.95, 111.272, -16.884, -82.745, 51.164]
  Set speed (120.0 mm/s)
  MoveL 8127 to (499.42, 509.32, 16.2) mm, rotated rx 0 ry 90 rz 0 deg; joints [-12.872, -27.972, 111.41, -16.904, -82.857, 51.132]
  Set speed (30.0 mm/s)
  Call Extruder(0.360)
  MoveL 8128 to (490.68, 500.58, 16.2) mm, rotated rx 0 ry 90 rz 0 deg; joints [-12.247, -28.165, 112.679, -16.239, -83.869, 50.76]
  Set speed (120.0 mm/s)
  MoveL 8129 to (490.68, 499.42, 16.2) mm, rotated rx 0 ry 90 rz 0 deg; joints [-12.139, -28.169, 112.709, -16.13, -83.891, 50.743]
  Set speed (30.0 mm/s)
  Call Extruder(0.360)
  MoveL 8130 to (499.42, 490.68, 16.2) mm, rotated rx 0 ry 90 rz 0 deg; joints [-11.163, -28.046, 111.884, -15.17, -83.189, 50.838]
  Set speed (120.0 mm/s)
  MoveL 8131 to (500.58, 490.68, 16.2) mm, rotated rx 0 ry 90 rz 0 deg; joints [-11.142, -28.025, 111.745, -15.152, -83.075, 50.866]
  Set speed (30.0 mm/s)
  Call Extruder(0.050)
  MoveL 8132 to (501.79, 491.89, 16.2) mm, rotated rx 0 ry 90 rz 0 deg; joints [-11.231, -27.997, 111.572, -15.246, -82.937, 50.915]
  Set speed (120.0 mm/s)
  MoveL 8133 to (502.08, 492.18, 16.2) mm, rotated rx 0 ry 90 rz 0 deg; joints [-11.252, -27.991, 111.53, -15.269, -82.903, 50.926]
  Set speed (30.0 mm/s)
  Call Extruder(0.298)
  MoveL 8134 to (509.32, 499.42, 16.2) mm, rotated rx 0 ry 90 rz 0 deg; joints [-11.777, -27.82, 110.483, -15.829, -82.076, 51.225]
  Set speed (120.0 mm/s)
  MoveL 8135 to (509.32, 500.58, 16.2) mm, rotated rx 0 ry 90 rz 0 deg; joints [-11.882, -27.815, 110.453, -15.936, -82.056, 51.244]
  Set speed (30.0 mm/s)
  Call Extruder(0.055)
  MoveL 8136 to (507.97, 501.92, 16.2) mm, rotated rx 0 ry 90 rz 0 deg; joints [-12.029, -27.836, 110.581, -16.08, -82.163, 51.233]
  MoveL 8137 to (507.85, 502.05, 16.2) mm, rotated rx 0 ry 90 rz 0 deg; joints [-12.043, -27.838, 110.593, -16.094, -82.173, 51.232]
  Set speed (120.0 mm/s)
  MoveL 8138 to (509.32, 490.68, 16.2) mm, rotated rx 0 ry 90 rz 0 deg; joints [-10.985, -27.855, 110.695, -15.024, -82.22, 51.08]
  Set speed (30.0 mm/s)
  Call Extruder(0.767)
  MoveL 8139 to (490.68, 509.32, 16.2) mm, rotated rx 0 ry 90 rz 0 deg; joints [-13.056, -28.131, 112.447, -17.059, -83.702, 50.893]
  MoveL 8140 to (490.56, 509.44, 16.2) mm, rotated rx 0 ry 90 rz 0 deg; joints [-13.07, -28.133, 112.458, -17.073, -83.712, 50.892]
  Set speed (120.0 mm/s)
  MoveL 8141 to (490.4, 509.6, 16.2) mm, rotated rx 0 ry 90 rz 0 deg; joints [-13.088, -28.135, 112.472, -17.091, -83.724, 50.89]
  Set speed (15.0 mm/s)
  Call Extruder(0.559)
  MoveL 8142 to (490.4, 490.4, 16.2) mm, rotated rx 0 ry 90 rz 0 deg; joints [-11.303, -28.206, 112.963, -15.284, -84.079, 50.608]
  MoveL 8143 to (509.6, 490.4, 16.2) mm, rotated rx 0 ry 90 rz 0 deg; joints [-10.955, -27.851, 110.668, -14.994, -82.197, 51.082]
  MoveL 8144 to (509.6, 509.6, 16.2) mm, rotated rx 0 ry 90 rz 0 deg; joints [-12.688, -27.769, 110.183, -16.759, -81.87, 51.41]
  MoveL 8145 to (490.4, 509.6, 16.2) mm, rotated rx 0 ry 90 rz 0 deg; joints [-13.088, -28.135, 112.472, -17.091, -83.724, 50.89]
  Set speed (120.0 mm/s)
  MoveL 8146 to (490.4, 509.2, 16.2) mm, rotated rx 0 ry 90 rz 0 deg; joints [-13.051, -28.136, 112.483, -17.053, -83.732, 50.884]
  Set speed (1000.0 mm/s)
  MoveL 8147 to (490.5, 509.2, 16.2) mm, rotated rx 0 ry 90 rz 0 deg; joints [-13.049, -28.135, 112.472, -17.051, -83.722, 50.886]
  Set speed (1000.0 mm/s)
  MoveL 8148 to (494.92, 492.25, 16.2) mm, rotated rx 0 ry 90 rz 0 deg; joints [-11.391, -28.122, 112.383, -15.387, -83.604, 50.748]
  Set speed (15.0 mm/s)
  Call Extruder(0.034)
  MoveL 8149 to (494.92, 491.09, 16.2) mm, rotated rx 0 ry 90 rz 0 deg; joints [-11.283, -28.126, 112.411, -15.277, -83.624, 50.732]
  Call Extruder(0.079)
  MoveL 8150 to (497.63, 491.09, 16.2) mm, rotated rx 0 ry 90 rz 0 deg; joints [-11.233, -28.077, 112.088, -15.235, -83.358, 50.799]
  Call Extruder(0.034)
  MoveL 8151 to (497.62, 492.26, 16.2) mm, rotated rx 0 ry 90 rz 0 deg; joints [-11.342, -28.073, 112.061, -15.345, -83.338, 50.817]
  Call Extruder(0.077)
  MoveL 8152 to (494.97, 492.26, 16.2) mm, rotated rx 0 ry 90 rz 0 deg; joints [-11.391, -28.121, 112.376, -15.387, -83.598, 50.75]
  Call Extruder(0.000)
  MoveL 8153 to (494.97, 492.25, 16.2) mm, rotated rx 0 ry 90 rz 0 deg; joints [-11.39, -28.121, 112.376, -15.386, -83.598, 50.75]
  Call Extruder(0.002)
  MoveL 8154 to (494.92, 492.25, 16.2) mm, rotated rx 0 ry 90 rz 0 deg; joints [-11.391, -28.122, 112.383, -15.387, -83.604, 50.748]
  Set speed (120.0 mm/s)
  MoveL 8155 to (495.23, 491.75, 16.2) mm, rotated rx 0 ry 90 rz 0 deg; joints [-11.339, -28.118, 112.358, -15.334, -83.581, 50.749]
  Set speed (15.0 mm/s)
  Call Extruder(0.014)
  MoveL 8156 to (495.57, 491.4, 16.2) mm, rotated rx 0 ry 90 rz 0 deg; joints [-11.3, -28.113, 112.325, -15.297, -83.554, 50.753]
  Set speed (120.0 mm/s)
  MoveL 8157 to (496.02, 491.95, 16.2) mm, rotated rx 0 ry 90 rz 0 deg; joints [-11.342, -28.103, 112.259, -15.34, -83.501, 50.772]
  Set speed (15.0 mm/s)
  Call Extruder(0.022)
  MoveL 8158 to (496.56, 491.4, 16.2) mm, rotated rx 0 ry 90 rz 0 deg; joints [-11.282, -28.095, 112.207, -15.281, -83.457, 50.777]
  Set speed (120.0 mm/s)
  MoveL 8159 to (497.01, 491.95, 16.2) mm, rotated rx 0 ry 90 rz 0 deg; joints [-11.324, -28.085, 112.141, -15.325, -83.403, 50.797]
  Set speed (15.0 mm/s)
  Call Extruder(0.012)
  MoveL 8160 to (497.31, 491.65, 16.2) mm, rotated rx 0 ry 90 rz 0 deg; joints [-11.291, -28.081, 112.113, -15.293, -83.379, 50.8]
  Set speed (120.0 mm/s)
  MoveL 8161 to (501.71, 491.09, 16.2) mm, rotated rx 0 ry 90 rz 0 deg; joints [-11.159, -28.002, 111.6, -15.173, -82.958, 50.9]
  Set speed (15.0 mm/s)
  Call Extruder(0.080)
  MoveL 8162 to (504.46, 491.09, 16.2) mm, rotated rx 0 ry 90 rz 0 deg; joints [-11.109, -27.949, 111.271, -15.132, -82.688, 50.968]
  Call Extruder(0.034)
  MoveL 8163 to (504.46, 492.27, 16.2) mm, rotated rx 0 ry 90 rz 0 deg; joints [-11.217, -27.945, 111.243, -15.242, -82.669, 50.986]
  Call Extruder(0.016)
  MoveL 8164 to (503.92, 492.26, 16.2) mm, rotated rx 0 ry 90 rz 0 deg; joints [-11.226, -27.955, 111.307, -15.249, -82.722, 50.973]
  Call Extruder(0.064)
  MoveL 8165 to (501.71, 492.26, 16.2) mm, rotated rx 0 ry 90 rz 0 deg; joints [-11.266, -27.997, 111.572, -15.282, -82.938, 50.918]
  Call Extruder(0.034)
  MoveL 8166 to (501.71, 491.09, 16.2) mm, rotated rx 0 ry 90 rz 0 deg; joints [-11.159, -28.002, 111.6, -15.173, -82.958, 50.9]
  Set speed (120.0 mm/s)
  MoveL 8167 to (502.02, 491.88, 16.2) mm, rotated rx 0 ry 90 rz 0 deg; joints [-11.226, -27.993, 111.544, -15.242, -82.914, 50.92]
  Set speed (15.0 mm/s)
  Call Extruder(0.020)
  MoveL 8168 to (502.5, 491.4, 16.2) mm, rotated rx 0 ry 90 rz 0 deg; joints [-11.173, -27.986, 111.498, -15.191, -82.875, 50.925]
  Set speed (120.0 mm/s)
  MoveL 8169 to (502.95, 491.95, 16.2) mm, rotated rx 0 ry 90 rz 0 deg; joints [-11.215, -27.975, 111.431, -15.234, -82.822, 50.944]
  Set speed (15.0 mm/s)
  Call Extruder(0.022)
  MoveL 8170 to (503.49, 491.4, 16.2) mm, rotated rx 0 ry 90 rz 0 deg; joints [-11.155, -27.967, 111.379, -15.176, -82.778, 50.949]
  Set speed (120.0 mm/s)
  MoveL 8171 to (503.94, 491.95, 16.2) mm, rotated rx 0 ry 90 rz 0 deg; joints [-11.197, -27.956, 111.313, -15.22, -82.725, 50.969]
  Set speed (15.0 mm/s)
  Call Extruder(0.008)
  MoveL 8172 to (504.14, 491.75, 16.2) mm, rotated rx 0 ry 90 rz 0 deg; joints [-11.175, -27.953, 111.293, -15.198, -82.709, 50.97]
  Set speed (120.0 mm/s)
  MoveL 8173 to (507.71, 494.38, 16.2) mm, rotated rx 0 ry 90 rz 0 deg; joints [-11.351, -27.873, 110.8, -15.389, -82.316, 51.101]
  Set speed (15.0 mm/s)
  Call Extruder(0.035)
  MoveL 8174 to (508.91, 494.38, 16.2) mm, rotated rx 0 ry 90 rz 0 deg; joints [-11.328, -27.849, 110.656, -15.371, -82.2, 51.13]
  Call Extruder(0.082)
  MoveL 8175 to (508.91, 497.19, 16.2) mm, rotated rx 0 ry 90 rz 0 deg; joints [-11.583, -27.837, 110.587, -15.631, -82.153, 51.177]
  Call Extruder(0.035)
  MoveL 8176 to (507.71, 497.19, 16.2) mm, rotated rx 0 ry 90 rz 0 deg; joints [-11.606, -27.861, 110.732, -15.649, -82.27, 51.147]
  Call Extruder(0.051)
  MoveL 8177 to (507.71, 495.45, 16.2) mm, rotated rx 0 ry 90 rz 0 deg; joints [-11.447, -27.868, 110.774, -15.488, -82.299, 51.118]
  Call Extruder(0.031)
  MoveL 8178 to (507.71, 494.38, 16.2) mm, rotated rx 0 ry 90 rz 0 deg; joints [-11.351, -27.873, 110.8, -15.389, -82.316, 51.101]
  Set speed (120.0 mm/s)
  MoveL 8179 to (508.59, 495.21, 16.2) mm, rotated rx 0 ry 90 rz 0 deg; joints [-11.41, -27.852, 110.674, -15.453, -82.217, 51.136]
  Set speed (15.0 mm/s)
  Call Extruder(0.023)
  MoveL 8180 to (508.03, 495.78, 16.2) mm, rotated rx 0 ry 90 rz 0 deg; joints [-11.472, -27.861, 110.729, -15.514, -82.263, 51.131]
  Set speed (120.0 mm/s)
  MoveL 8181 to (508.59, 496.2, 16.2) mm, rotated rx 0 ry 90 rz 0 deg; joints [-11.5, -27.848, 110.65, -15.544, -82.2, 51.152]
  Set speed (15.0 mm/s)
  Call Extruder(0.023)
  MoveL 8182 to (508.03, 496.77, 16.2) mm, rotated rx 0 ry 90 rz 0 deg; joints [-11.562, -27.857, 110.704, -15.605, -82.246, 51.148]
  Set speed (120.0 mm/s)
  MoveL 8183 to (507.71, 501.84, 16.2) mm, rotated rx 0 ry 90 rz 0 deg; joints [-12.027, -27.842, 110.615, -16.077, -82.19, 51.225]
  Set speed (15.0 mm/s)
  Call Extruder(0.035)
  MoveL 8184 to (508.91, 501.85, 16.2) mm, rotated rx 0 ry 90 rz 0 deg; joints [-12.004, -27.818, 110.47, -16.059, -82.074, 51.255]
  Call Extruder(0.082)
  MoveL 8185 to (508.91, 504.67, 16.2) mm, rotated rx 0 ry 90 rz 0 deg; joints [-12.259, -27.805, 110.397, -16.318, -82.025, 51.304]
  Call Extruder(0.035)
  MoveL 8186 to (507.71, 504.67, 16.2) mm, rotated rx 0 ry 90 rz 0 deg; joints [-12.282, -27.83, 110.542, -16.337, -82.141, 51.273]
  Call Extruder(0.082)
  MoveL 8187 to (507.71, 501.84, 16.2) mm, rotated rx 0 ry 90 rz 0 deg; joints [-12.027, -27.842, 110.615, -16.077, -82.19, 51.225]
  Set speed (120.0 mm/s)
  MoveL 8188 to (508.58, 502.16, 16.2) mm, rotated rx 0 ry 90 rz 0 deg; joints [-12.039, -27.823, 110.502, -16.093, -82.101, 51.252]
  Set speed (15.0 mm/s)
  Call Extruder(0.023)
  MoveL 8189 to (508.03, 502.71, 16.2) mm, rotated rx 0 ry 90 rz 0 deg; joints [-12.099, -27.832, 110.555, -16.152, -82.145, 51.248]
  Set speed (120.0 mm/s)
  MoveL 8190 to (508.59, 503.13, 16.2) mm, rotated rx 0 ry 90 rz 0 deg; joints [-12.126, -27.818, 110.475, -16.182, -82.082, 51.27]
  Set speed (15.0 mm/s)
  Call Extruder(0.023)
  MoveL 8191 to (508.02, 503.7, 16.2) mm, rotated rx 0 ry 90 rz 0 deg; joints [-12.189, -27.828, 110.529, -16.243, -82.127, 51.265]
  Set speed (120.0 mm/s)
  MoveL 8192 to (508.59, 504.12, 16.2) mm, rotated rx 0 ry 90 rz 0 deg; joints [-12.216, -27.814, 110.45, -16.273, -82.065, 51.287]
  Set speed (15.0 mm/s)
  Call Extruder(0.010)
  MoveL 8193 to (508.36, 504.36, 16.2) mm, rotated rx 0 ry 90 rz 0 deg; joints [-12.241, -27.818, 110.472, -16.298, -82.083, 51.285]
  Set speed (120.0 mm/s)
  MoveL 8194 to (490.68, 490.68, 16.2) mm, rotated rx 0 ry 90 rz 0 deg; joints [-11.324, -28.2, 112.923, -15.306, -84.047, 50.619]
  Set speed (1000.0 mm/s)
  MoveL 8195 to (490.68, 490.68, 16.3) mm, rotated rx 0 ry 90 rz 0 deg; joints [-11.324, -28.211, 112.929, -15.306, -84.042, 50.621]
  Set speed (30.0 mm/s)
  Call Extruder(0.767)
  MoveL 8196 to (509.32, 509.32, 16.3) mm, rotated rx 0 ry 90 rz 0 deg; joints [-12.669, -27.786, 110.229, -16.738, -81.897, 51.399]
  MoveL 8197 to (509.44, 509.44, 16.3) mm, rotated rx 0 ry 90 rz 0 deg; joints [-12.677, -27.783, 110.211, -16.747, -81.883, 51.404]
  Set speed (120.0 mm/s)
  MoveL 8198 to (507.79, 502.11, 16.3) mm, rotated rx 0 ry 90 rz 0 deg; joints [-12.049, -27.85, 110.604, -16.1, -82.173, 51.233]
  Set speed (30.0 mm/s)
  Call Extruder(0.297)
  MoveL 8199 to (500.58, 509.32, 16.3) mm, rotated rx 0 ry 90 rz 0 deg; joints [-12.847, -27.96, 111.277, -16.884, -82.74, 51.165]
  Set speed (120.0 mm/s)
  MoveL 8200 to (499.42, 509.32, 16.3) mm, rotated rx 0 ry 90 rz 0 deg; joints [-12.872, -27.982, 111.416, -16.904, -82.852, 51.134]
  Set speed (30.0 mm/s)
  Call Extruder(0.360)
  MoveL 8201 to (490.68, 500.58, 16.3) mm, rotated rx 0 ry 90 rz 0 deg; joints [-12.247, -28.176, 112.684, -16.239, -83.864, 50.762]
  Set speed (120.0 mm/s)
  MoveL 8202 to (490.68, 499.42, 16.3) mm, rotated rx 0 ry 90 rz 0 deg; joints [-12.139, -28.18, 112.714, -16.13, -83.885, 50.745]
  Set speed (30.0 mm/s)
  MoveL 8203 to (499.42, 490.68, 16.3) mm, rotated rx 0 ry 90 rz 0 deg; joints [-11.163, -28.057, 111.889, -15.17, -83.184, 50.839]
  Set speed (120.0 mm/s)
  MoveL 8204 to (500.58, 490.68, 16.3) mm, rotated rx 0 ry 90 rz 0 deg; joints [-11.141, -28.035, 111.75, -15.152, -83.07, 50.868]
  Set speed (30.0 mm/s)
  Call Extruder(0.052)
  MoveL 8205 to (501.85, 491.95, 16.3) mm, rotated rx 0 ry 90 rz 0 deg; joints [-11.235, -28.007, 111.568, -15.252, -82.924, 50.919]
  Set speed (120.0 mm/s)
  MoveL 8206 to (502.08, 492.18, 16.3) mm, rotated rx 0 ry 90 rz 0 deg; joints [-11.252, -28.001, 111.535, -15.269, -82.898, 50.928]
  Set speed (30.0 mm/s)
  Call Extruder(0.298)
  MoveL 8207 to (509.32, 499.42, 16.3) mm, rotated rx 0 ry 90 rz 0 deg; joints [-11.777, -27.83, 110.488, -15.83, -82.071, 51.226]
  Set speed (120.0 mm/s)
  MoveL 8208 to (509.32, 500.58, 16.3) mm, rotated rx 0 ry 90 rz 0 deg; joints [-11.882, -27.825, 110.458, -15.936, -82.051, 51.246]
  Set speed (30.0 mm/s)
  Call Extruder(0.058)
  MoveL 8209 to (507.92, 501.98, 16.3) mm, rotated rx 0 ry 90 rz 0 deg; joints [-12.035, -27.848, 110.591, -16.086, -82.163, 51.234]
  MoveL 8210 to (507.8, 502.1, 16.3) mm, rotated rx 0 ry 90 rz 0 deg; joints [-12.049, -27.85, 110.603, -16.1, -82.172, 51.233]
  Set speed (120.0 mm/s)
  MoveL 8211 to (509.32, 490.68, 16.3) mm, rotated rx 0 ry 90 rz 0 deg; joints [-10.985, -27.866, 110.7, -15.024, -82.214, 51.081]
  Set speed (30.0 mm/s)
  Call Extruder(0.767)
  MoveL 8212 to (490.68, 509.32, 16.3) mm, rotated rx 0 ry 90 rz 0 deg; joints [-13.056, -28.142, 112.452, -17.059, -83.697, 50.895]
  MoveL 8213 to (490.56, 509.44, 16.3) mm, rotated rx 0 ry 90 rz 0 deg; joints [-13.07, -28.143, 112.464, -17.073, -83.707, 50.893]
  Set speed (120.0 mm/s)
  MoveL 8214 to (490.4, 509.6, 16.3) mm, rotated rx 0 ry 90 rz 0 deg; joints [-13.088, -28.145, 112.478, -17.091, -83.719, 50.891]
  Set speed (15.0 mm/s)
  Call Extruder(0.559)
  MoveL 8215 to (490.4, 490.4, 16.3) mm, rotated rx 0 ry 90 rz 0 deg; joints [-11.303, -28.217, 112.968, -15.284, -84.074, 50.61]
  MoveL 8216 to (509.6, 490.4, 16.3) mm, rotated rx 0 ry 90 rz 0 deg; joints [-10.955, -27.861, 110.673, -14.994, -82.191, 51.084]
  MoveL 8217 to (509.6, 509.6, 16.3) mm, rotated rx 0 ry 90 rz 0 deg; joints [-12.688, -27.779, 110.188, -16.759, -81.865, 51.411]
  MoveL 8218 to (490.4, 509.6, 16.3) mm, rotated rx 0 ry 90 rz 0 deg; joints [-13.088, -28.145, 112.478, -17.091, -83.719, 50.891]
  Set speed (120.0 mm/s)
  MoveL 8219 to (490.4, 509.2, 16.3) mm, rotated rx 0 ry 90 rz 0 deg; joints [-13.051, -28.147, 112.489, -17.053, -83.726, 50.885]
  Set speed (1000.0 mm/s)
  MoveL 8220 to (490.5, 509.2, 16.3) mm, rotated rx 0 ry 90 rz 0 deg; joints [-13.049, -28.145, 112.477, -17.051, -83.717, 50.888]
  Set speed (1000.0 mm/s)
  MoveL 8221 to (494.92, 492.25, 16.3) mm, rotated rx 0 ry 90 rz 0 deg; joints [-11.391, -28.132, 112.388, -15.387, -83.598, 50.75]
  Set speed (15.0 mm/s)
  Call Extruder(0.034)
  MoveL 8222 to (494.92, 491.09, 16.3) mm, rotated rx 0 ry 90 rz 0 deg; joints [-11.283, -28.136, 112.416, -15.277, -83.618, 50.733]
  Call Extruder(0.077)
  MoveL 8223 to (497.57, 491.09, 16.3) mm, rotated rx 0 ry 90 rz 0 deg; joints [-11.234, -28.089, 112.1, -15.236, -83.358, 50.799]
  Call Extruder(0.034)
  MoveL 8224 to (497.57, 492.26, 16.3) mm, rotated rx 0 ry 90 rz 0 deg; joints [-11.343, -28.085, 112.072, -15.346, -83.338, 50.817]
  Call Extruder(0.076)
  MoveL 8225 to (494.97, 492.26, 16.3) mm, rotated rx 0 ry 90 rz 0 deg; joints [-11.391, -28.131, 112.381, -15.387, -83.593, 50.751]
  Call Extruder(0.000)
  MoveL 8226 to (494.97, 492.25, 16.3) mm, rotated rx 0 ry 90 rz 0 deg; joints [-11.39, -28.131, 112.382, -15.386, -83.593, 50.751]
  Call Extruder(0.002)
  MoveL 8227 to (494.92, 492.25, 16.3) mm, rotated rx 0 ry 90 rz 0 deg; joints [-11.391, -28.132, 112.388, -15.387, -83.598, 50.75]
  Set speed (120.0 mm/s)
  MoveL 8228 to (495.37, 491.41, 16.3) mm, rotated rx 0 ry 90 rz 0 deg; joints [-11.304, -28.127, 112.355, -15.3, -83.569, 50.749]
  Set speed (15.0 mm/s)
  Call Extruder(0.022)
  MoveL 8229 to (495.91, 491.95, 16.3) mm, rotated rx 0 ry 90 rz 0 deg; joints [-11.344, -28.116, 112.278, -15.342, -83.507, 50.77]
  Set speed (120.0 mm/s)
  MoveL 8230 to (496.36, 491.4, 16.3) mm, rotated rx 0 ry 90 rz 0 deg; joints [-11.286, -28.11, 112.237, -15.285, -83.472, 50.774]
  Set speed (15.0 mm/s)
  MoveL 8231 to (496.9, 491.95, 16.3) mm, rotated rx 0 ry 90 rz 0 deg; joints [-11.326, -28.098, 112.16, -15.327, -83.41, 50.795]
  Set speed (120.0 mm/s)
  MoveL 8232 to (501.77, 492.26, 16.3) mm, rotated rx 0 ry 90 rz 0 deg; joints [-11.265, -28.007, 111.57, -15.282, -82.927, 50.921]
  Set speed (15.0 mm/s)
  Call Extruder(0.034)
  MoveL 8233 to (501.77, 491.09, 16.3) mm, rotated rx 0 ry 90 rz 0 deg; joints [-11.158, -28.011, 111.598, -15.172, -82.946, 50.903]
  Call Extruder(0.078)
  MoveL 8234 to (504.46, 491.09, 16.3) mm, rotated rx 0 ry 90 rz 0 deg; joints [-11.109, -27.96, 111.276, -15.133, -82.683, 50.969]
  Call Extruder(0.034)
  MoveL 8235 to (504.46, 492.27, 16.3) mm, rotated rx 0 ry 90 rz 0 deg; joints [-11.217, -27.956, 111.248, -15.242, -82.664, 50.988]
  Call Extruder(0.016)
  MoveL 8236 to (503.92, 492.26, 16.3) mm, rotated rx 0 ry 90 rz 0 deg; joints [-11.226, -27.966, 111.312, -15.249, -82.716, 50.975]
  Call Extruder(0.063)
  MoveL 8237 to (501.77, 492.26, 16.3) mm, rotated rx 0 ry 90 rz 0 deg; joints [-11.265, -28.007, 111.57, -15.282, -82.927, 50.921]
  Set speed (120.0 mm/s)
  MoveL 8238 to (502.29, 491.4, 16.3) mm, rotated rx 0 ry 90 rz 0 deg; joints [-11.177, -28, 111.528, -15.194, -82.89, 50.921]
  Set speed (15.0 mm/s)
  Call Extruder(0.022)
  MoveL 8239 to (502.84, 491.95, 16.3) mm, rotated rx 0 ry 90 rz 0 deg; joints [-11.217, -27.988, 111.45, -15.236, -82.828, 50.943]
  Set speed (120.0 mm/s)
  MoveL 8240 to (503.28, 491.4, 16.3) mm, rotated rx 0 ry 90 rz 0 deg; joints [-11.159, -27.981, 111.409, -15.179, -82.793, 50.945]
  Set speed (15.0 mm/s)
  Call Extruder(0.022)
  MoveL 8241 to (503.83, 491.95, 16.3) mm, rotated rx 0 ry 90 rz 0 deg; joints [-11.199, -27.969, 111.332, -15.221, -82.731, 50.967]
  Set speed (120.0 mm/s)
  MoveL 8242 to (507.72, 494.39, 16.3) mm, rotated rx 0 ry 90 rz 0 deg; joints [-11.351, -27.883, 110.805, -15.39, -82.311, 51.102]
  Set speed (15.0 mm/s)
  Call Extruder(0.035)
  MoveL 8243 to (508.91, 494.38, 16.3) mm, rotated rx 0 ry 90 rz 0 deg; joints [-11.328, -27.859, 110.661, -15.371, -82.195, 51.132]
  Call Extruder(0.080)
  MoveL 8244 to (508.91, 497.13, 16.3) mm, rotated rx 0 ry 90 rz 0 deg; joints [-11.578, -27.848, 110.594, -15.626, -82.149, 51.177]
  Call Extruder(0.035)
  MoveL 8245 to (507.71, 497.14, 16.3) mm, rotated rx 0 ry 90 rz 0 deg; joints [-11.6, -27.872, 110.738, -15.644, -82.265, 51.147]
  Call Extruder(0.051)
  MoveL 8246 to (507.71, 495.39, 16.3) mm, rotated rx 0 ry 90 rz 0 deg; joints [-11.442, -27.879, 110.781, -15.482, -82.294, 51.119]
  Call Extruder(0.029)
  MoveL 8247 to (507.72, 494.39, 16.3) mm, rotated rx 0 ry 90 rz 0 deg; joints [-11.351, -27.883, 110.805, -15.39, -82.311, 51.102]
  Set speed (120.0 mm/s)
  MoveL 8248 to (508.03, 495.16, 16.3) mm, rotated rx 0 ry 90 rz 0 deg; joints [-11.415, -27.874, 110.749, -15.456, -82.268, 51.123]
  Set speed (15.0 mm/s)
  Call Extruder(0.023)
  MoveL 8249 to (508.59, 495.72, 16.3) mm, rotated rx 0 ry 90 rz 0 deg; joints [-11.456, -27.86, 110.667, -15.5, -82.203, 51.146]
  Set speed (120.0 mm/s)
  MoveL 8250 to (508.03, 496.15, 16.3) mm, rotated rx 0 ry 90 rz 0 deg; joints [-11.505, -27.87, 110.725, -15.548, -82.251, 51.139]
  Set speed (15.0 mm/s)
  Call Extruder(0.023)
  MoveL 8251 to (508.59, 496.71, 16.3) mm, rotated rx 0 ry 90 rz 0 deg; joints [-11.546, -27.856, 110.642, -15.591, -82.187, 51.162]
  Set speed (120.0 mm/s)
